KUKA KRL program: MyProgram_221().src

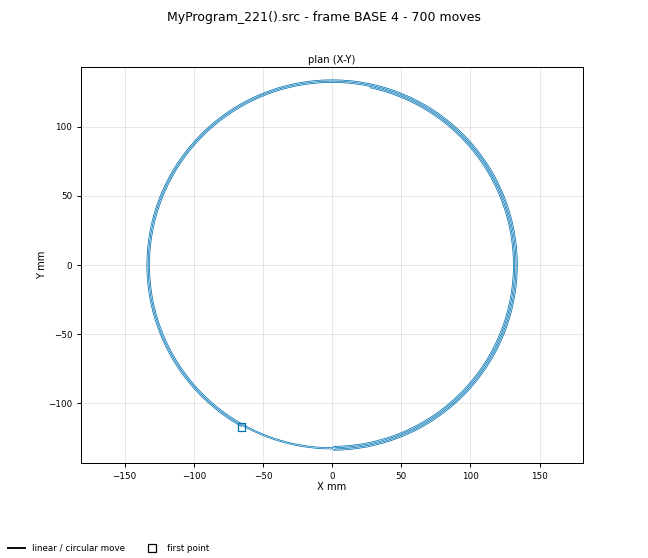
[picture p0: tool path of MyProgram_221().src in frame BASE 4, 700 of 700 moves have a stored position in this frame; points joined in program order, loops and branches not executed]
&ACCESS RVP
&REL 1
&PARAM TEMPLATE = C:\KRC\Roboter\Template\vorgabe
&PARAM EDITMASK = *
DEF MyProgram_221()
; ---- Setting reference (Base) ----
$BASE = BASE_DATA[4]

; --------------------------
; ---- Setting tool (TCP) ----
$TOOL = TOOL_DATA[3]
; --------------------------

$VEL.CP = VEL_APROX_PRINT
Startdeposition()
$VEL.CP = VEL_PRINT
LIN {X -65.4764,Y -116.7395,Z 154,A -122.5676,B 24.2106,C -1.1477,E1 24.1569,E2 209.4417} C_DIS
LIN {X -69.4702,Y -114.408,Z 154,A -124.5396,B 24.2105,C -1.151,E1 24.1522,E2 211.4118} C_DIS
LIN {X -73.2404,Y -112.0324,Z 154,A -126.4311,B 24.2103,C -1.1548,E1 24.1478,E2 213.3004} C_DIS
LIN {X -76.6718,Y -109.7121,Z 154,A -128.2386,B 24.2103,C -1.1561,E1 24.1436,E2 215.111} C_DIS
LIN {X -80.258,Y -107.117,Z 154,A -130.1581,B 24.2101,C -1.1583,E1 24.1393,E2 217.0323} C_DIS
LIN {X -83.7739,Y -104.39,Z 154,A -132.0662,B 24.21,C -1.1616,E1 24.1351,E2 218.9394} C_DIS
LIN {X -87.1638,Y -101.5764,Z 154,A -133.9639,B 24.2098,C -1.1647,E1 24.131,E2 220.837} C_DIS
LIN {X -90.549,Y -98.5704,Z 154,A -136.3247,B 24.2106,C -1.1484,E1 24.1261,E2 223.2477} C_DIS
LIN {X -93.7846,Y -95.4971,Z 154,A -138.0959,B 24.2101,C -1.1591,E1 24.1226,E2 225.0003} C_DIS
LIN {X -96.4017,Y -92.8551,Z 154,A -139.4034,B 24.2093,C -1.1762,E1 24.1201,E2 226.2717} C_DIS
LIN {X -99.4158,Y -89.621,Z 154,A -141.3271,B 24.2092,C -1.179,E1 24.1165,E2 228.1973} C_DIS
LIN {X -102.4018,Y -86.1925,Z 154,A -143.0746,B 24.2085,C -1.1931,E1 24.1133,E2 229.9185} C_DIS
LIN {X -107.1454,Y -80.2198,Z 154,A -146.5875,B 24.2087,C -1.1892,E1 24.1072,E2 233.4581} C_DIS
LIN {X -109.8326,Y -76.4986,Z 154,A -148.5307,B 24.2084,C -1.1953,E1 24.1041,E2 235.3964} C_DIS
LIN {X -112.3217,Y -72.7948,Z 154,A -150.4236,B 24.2082,C -1.2011,E1 24.1012,E2 237.2849} C_DIS
LIN {X -114.6316,Y -69.1005,Z 154,A -152.3129,B 24.208,C -1.2049,E1 24.0984,E2 239.1748} C_DIS
LIN {X -116.8933,Y -65.2026,Z 154,A -154.2587,B 24.2078,C -1.2094,E1 24.0957,E2 241.12} C_DIS
LIN {X -118.9758,Y -61.3183,Z 154,A -156.1666,B 24.2076,C -1.2137,E1 24.0933,E2 243.0279} C_DIS
LIN {X -120.9571,Y -57.3088,Z 154,A -158.0095,B 24.2072,C -1.2226,E1 24.091,E2 244.8594} C_DIS
LIN {X -122.9724,Y -52.8453,Z 154,A -160.0801,B 24.2068,C -1.2299,E1 24.0887,E2 246.9239} C_DIS
LIN {X -124.2089,Y -49.8691,Z 154,A -161.4613,B 24.2066,C -1.2339,E1 24.0872,E2 248.3033} C_DIS
LIN {X -125.3493,Y -46.9286,Z 154,A -162.8567,B 24.2066,C -1.2358,E1 24.0858,E2 249.702} C_DIS
LIN {X -126.5669,Y -43.5392,Z 154,A -164.3642,B 24.2062,C -1.2421,E1 24.0844,E2 251.2031} C_DIS
LIN {X -127.5513,Y -40.5643,Z 154,A -165.7297,B 24.2061,C -1.2451,E1 24.0833,E2 252.5694} C_DIS
LIN {X -128.4924,Y -37.4767,Z 154,A -167.1511,B 24.206,C -1.2475,E1 24.0821,E2 253.9935} C_DIS
LIN {X -129.5708,Y -33.5652,Z 154,A -169.0376,B 24.206,C -1.2458,E1 24.0807,E2 255.8954} C_DIS
LIN {X -130.5475,Y -29.5336,Z 154,A -170.6264,B 24.2054,C -1.2602,E1 24.0797,E2 257.4585} C_DIS
LIN {X -131.1874,Y -26.546,Z 154,A -172.5665,B 24.2066,C -1.2349,E1 24.0786,E2 259.4727} C_DIS
LIN {X -132.0312,Y -21.968,Z 154,A -173.9924,B 24.205,C -1.2676,E1 24.078,E2 260.827} C_DIS
LIN {X -132.553,Y -18.5652,Z 154,A -175.5736,B 24.205,C -1.2673,E1 24.0773,E2 262.4186} C_DIS
LIN {X -133.0698,Y -14.3967,Z 154,A -177.3185,B 24.2046,C -1.2756,E1 24.0768,E2 264.154} C_DIS
LIN {X -133.4458,Y -10.3664,Z 154,A -179.1414,B 24.2046,C -1.277,E1 24.0763,E2 265.9848} C_DIS
LIN {X -133.6901,Y -6.4724,Z 154,A 179.2809,B 24.204,C -1.2868,E1 24.0761,E2 267.5484} C_DIS
LIN {X -133.8245,Y -2.4362,Z 154,A 177.4846,B 24.204,C -1.2893,E1 24.076,E2 269.3498} C_DIS
LIN {X -133.831,Y 2.0454,Z 154,A 175.6023,B 24.2035,C -1.2973,E1 24.076,E2 271.2242} C_DIS
LIN {X -133.7281,Y 5.6424,Z 154,A 173.9321,B 24.2035,C -1.2963,E1 24.0762,E2 272.9073} C_DIS
LIN {X -133.4911,Y 9.7453,Z 154,A 172.2639,B 24.2031,C -1.3063,E1 24.0765,E2 274.5613} C_DIS
LIN {X -133.1347,Y 13.7941,Z 154,A 170.4691,B 24.2029,C -1.3094,E1 24.0769,E2 276.3596} C_DIS
LIN {X -132.7029,Y 17.4579,Z 154,A 168.9226,B 24.2026,C -1.3162,E1 24.0775,E2 277.8992} C_DIS
LIN {X -132.1182,Y 21.4462,Z 154,A 166.9905,B 24.2028,C -1.3122,E1 24.0783,E2 279.8529} C_DIS
LIN {X -131.3493,Y 25.7398,Z 154,A 165.3027,B 24.202,C -1.3266,E1 24.0792,E2 281.5157} C_DIS
LIN {X -129.9408,Y 32.1056,Z 154,A 162.5341,B 24.2015,C -1.3367,E1 24.0809,E2 284.2764} C_DIS
LIN {X -128.8361,Y 36.2779,Z 154,A 160.6208,B 24.2013,C -1.3396,E1 24.0823,E2 286.1942} C_DIS
LIN {X -127.7534,Y 39.9286,Z 154,A 158.5002,B 24.2023,C -1.322,E1 24.0841,E2 288.3705} C_DIS
LIN {X -126.4374,Y 43.913,Z 154,A 157.192,B 24.2008,C -1.3503,E1 24.0852,E2 289.6168} C_DIS
LIN {X -125.2818,Y 47.1088,Z 154,A 155.7275,B 24.2006,C -1.3544,E1 24.0866,E2 291.0799} C_DIS
LIN {X -124.0765,Y 50.1976,Z 154,A 154.2876,B 24.2004,C -1.3579,E1 24.0881,E2 292.5196} C_DIS
LIN {X -122.5281,Y 53.8719,Z 154,A 152.4761,B 24.2004,C -1.3583,E1 24.0901,E2 294.3407} C_DIS
LIN {X -119.6547,Y 59.9846,Z 154,A 149.6779,B 24.1997,C -1.3714,E1 24.0935,E2 297.1224} C_DIS
LIN {X -117.7054,Y 63.7246,Z 154,A 147.8801,B 24.1994,C -1.3771,E1 24.0958,E2 298.9159} C_DIS
LIN {X -116.2233,Y 66.3882,Z 154,A 146.4488,B 24.1994,C -1.3751,E1 24.0978,E2 300.3601} C_DIS
LIN {X -113.8859,Y 70.3235,Z 154,A 144.4779,B 24.1992,C -1.3802,E1 24.1006,E2 302.3289} C_DIS
LIN {X -111.5508,Y 73.9718,Z 154,A 142.5696,B 24.1991,C -1.383,E1 24.1035,E2 304.2403} C_DIS
LIN {X -108.9939,Y 77.6892,Z 154,A 140.6453,B 24.1987,C -1.3887,E1 24.1066,E2 306.1603} C_DIS
LIN {X -106.2792,Y 81.3632,Z 154,A 138.6861,B 24.1985,C -1.3939,E1 24.1099,E2 308.1166} C_DIS
LIN {X -103.8356,Y 84.4601,Z 154,A 136.9688,B 24.1983,C -1.3971,E1 24.1129,E2 309.8344} C_DIS
LIN {X -101.0139,Y 87.8152,Z 154,A 134.9381,B 24.1984,C -1.3947,E1 24.1166,E2 311.8804} C_DIS
LIN {X -96.0669,Y 93.2009,Z 154,A 131.9703,B 24.1976,C -1.4103,E1 24.1222,E2 314.8235} C_DIS
LIN {X -91.6081,Y 97.5874,Z 154,A 129.3779,B 24.197,C -1.4208,E1 24.1274,E2 317.4014} C_DIS
LIN {X -87.1976,Y 101.5473,Z 154,A 126.7888,B 24.1968,C -1.4242,E1 24.1328,E2 319.9928} C_DIS
LIN {X -84.1281,Y 104.1044,Z 154,A 124.7816,B 24.1974,C -1.4139,E1 24.1372,E2 322.033} C_DIS
LIN {X -81.4973,Y 106.1766,Z 154,A 123.2234,B 24.1975,C -1.4111,E1 24.1407,E2 323.604} C_DIS
LIN {X -78.3223,Y 108.54,Z 154,A 121.9651,B 24.1962,C -1.4353,E1 24.1434,E2 324.8076} C_DIS
LIN {X -75.2508,Y 110.6916,Z 154,A 120.2271,B 24.1964,C -1.4323,E1 24.1474,E2 326.5593} C_DIS
LIN {X -71.4037,Y 113.2111,Z 154,A 118.2937,B 24.1961,C -1.4377,E1 24.152,E2 328.4856} C_DIS
LIN {X -67.5784,Y 115.5356,Z 154,A 116.3255,B 24.196,C -1.4388,E1 24.1567,E2 330.4575} C_DIS
LIN {X -63.6092,Y 117.7676,Z 154,A 114.4022,B 24.1957,C -1.4434,E1 24.1614,E2 332.3751} C_DIS
LIN {X -60.562,Y 119.3608,Z 154,A 113.0252,B 24.1953,C -1.4505,E1 24.1648,E2 333.7388} C_DIS
LIN {X -57.5921,Y 120.8217,Z 154,A 111.5955,B 24.1953,C -1.4521,E1 24.1683,E2 335.1682} C_DIS
LIN {X -54.4903,Y 122.2521,Z 154,A 110.1144,B 24.1952,C -1.4535,E1 24.1721,E2 336.6499} C_DIS
LIN {X -51.3156,Y 123.6185,Z 154,A 108.6293,B 24.1951,C -1.4553,E1 24.1759,E2 338.1339} C_DIS
LIN {X -48.2296,Y 124.8548,Z 154,A 107.2262,B 24.1949,C -1.4583,E1 24.1796,E2 339.533} C_DIS
LIN {X -45.123,Y 126.0109,Z 154,A 105.7967,B 24.1949,C -1.4596,E1 24.1833,E2 340.9623} C_DIS
LIN {X -42.0962,Y 127.054,Z 154,A 104.423,B 24.1947,C -1.4611,E1 24.1869,E2 342.3349} C_DIS
LIN {X -38.7731,Y 128.1077,Z 154,A 102.9369,B 24.1947,C -1.4631,E1 24.1909,E2 343.8188} C_DIS
LIN {X -35.6125,Y 129.0222,Z 154,A 101.3601,B 24.195,C -1.4564,E1 24.1952,E2 345.4146} C_DIS
LIN {X -31.458,Y 130.0969,Z 154,A 99.6528,B 24.1945,C -1.4646,E1 24.1998,E2 347.1044} C_DIS
LIN {X -28.1162,Y 130.8598,Z 154,A 98.2044,B 24.1945,C -1.4668,E1 24.2037,E2 348.5493} C_DIS
LIN {X -24.9126,Y 131.5075,Z 154,A 96.7704,B 24.1945,C -1.4663,E1 24.2076,E2 349.9864} C_DIS
LIN {X -20.8025,Y 132.2202,Z 154,A 94.9726,B 24.1945,C -1.4669,E1 24.2126,E2 351.7842} C_DIS
LIN {X -17.2485,Y 132.7303,Z 154,A 93.4692,B 24.1943,C -1.4696,E1 24.2167,E2 353.2824} C_DIS
LIN {X -13.434,Y 133.172,Z 154,A 91.7062,B 24.1945,C -1.4646,E1 24.2217,E2 355.0588} C_DIS
LIN {X -9.6554,Y 133.4977,Z 154,A 90.2127,B 24.1941,C -1.4717,E1 24.2258,E2 356.5354} C_DIS
LIN {X -6.0046,Y 133.7136,Z 154,A 88.4886,B 24.1945,C -1.4644,E1 24.2306,E2 358.2778} C_DIS
LIN {X -2.0508,Y 133.8309,Z 154,A 86.9521,B 24.1941,C -1.4727,E1 24.2349,E2 359.7943} C_DIS
LIN {X 1.6346,Y 133.8378,Z 154,A 85.2383,B 24.1944,C -1.4661,E1 24.2397,E2 361.5239} C_DIS
LIN {X 5.3279,Y 133.7404,Z 154,A 83.7365,B 24.1942,C -1.4703,E1 24.2439,E2 363.0153} C_DIS
LIN {X 9.5685,Y 133.504,Z 154,A 81.9349,B 24.1942,C -1.4711,E1 24.2489,E2 364.8142} C_DIS
LIN {X 13.162,Y 133.1981,Z 154,A 80.3288,B 24.1944,C -1.4678,E1 24.2534,E2 366.4274} C_DIS
LIN {X 17.2746,Y 132.7269,Z 154,A 78.6281,B 24.1942,C -1.471,E1 24.2581,E2 368.1188} C_DIS
LIN {X 20.8308,Y 132.2158,Z 154,A 76.9846,B 24.1945,C -1.4652,E1 24.2626,E2 369.7748} C_DIS
LIN {X 24.9827,Y 131.4941,Z 154,A 75.2937,B 24.1942,C -1.4702,E1 24.2672,E2 371.4517} C_DIS
LIN {X 28.3093,Y 130.8181,Z 154,A 73.8631,B 24.1942,C -1.4706,E1 24.2711,E2 372.8794} C_DIS
LIN {X 31.4122,Y 130.1079,Z 154,A 72.501,B 24.1942,C -1.4699,E1 24.2748,E2 374.2414} C_DIS
LIN {X 34.6166,Y 129.2922,Z 154,A 71.066,B 24.1943,C -1.468,E1 24.2787,E2 375.6786} C_DIS
LIN {X 38.4085,Y 128.2193,Z 154,A 69.405,B 24.1943,C -1.468,E1 24.2832,E2 377.3366} C_DIS
LIN {X 40.9294,Y 127.4346,Z 154,A 67.9832,B 24.1952,C -1.4523,E1 24.2871,E2 378.7939} C_DIS
LIN {X 45.0326,Y 126.0435,Z 154,A 66.3563,B 24.1947,C -1.4622,E1 24.2913,E2 380.3933} C_DIS
LIN {X 48.6514,Y 124.6909,Z 154,A 64.7453,B 24.1947,C -1.4628,E1 24.2955,E2 381.9994} C_DIS
LIN {X 51.8882,Y 123.3793,Z 154,A 63.2634,B 24.1947,C -1.4618,E1 24.2993,E2 383.48} C_DIS
LIN {X 54.8155,Y 122.1066,Z 154,A 61.9074,B 24.1947,C -1.4608,E1 24.3027,E2 384.8351} C_DIS
LIN {X 57.9391,Y 120.656,Z 154,A 60.4143,B 24.1949,C -1.458,E1 24.3065,E2 386.331} C_DIS
LIN {X 61.0008,Y 119.1374,Z 154,A 58.9467,B 24.195,C -1.4558,E1 24.3102,E2 387.7997} C_DIS
LIN {X 64.4312,Y 117.3201,Z 154,A 57.1908,B 24.1954,C -1.4487,E1 24.3145,E2 389.5679} C_DIS
LIN {X 68.3558,Y 115.0772,Z 154,A 55.2802,B 24.1955,C -1.447,E1 24.3191,E2 391.4764} C_DIS
LIN {X 72.1374,Y 112.745,Z 154,A 53.3962,B 24.1956,C -1.445,E1 24.3236,E2 393.3591} C_DIS
LIN {X 76.0047,Y 110.1754,Z 154,A 51.4174,B 24.1958,C -1.4421,E1 24.3282,E2 395.3381} C_DIS
LIN {X 79.603,Y 107.6047,Z 154,A 49.5047,B 24.1961,C -1.4377,E1 24.3325,E2 397.2545} C_DIS
LIN {X 83.1317,Y 104.9021,Z 154,A 47.6134,B 24.1962,C -1.4347,E1 24.3367,E2 399.1457} C_DIS
LIN {X 86.5146,Y 102.1299,Z 154,A 45.7441,B 24.1964,C -1.4312,E1 24.3407,E2 401.016} C_DIS
LIN {X 90.0812,Y 98.9983,Z 154,A 43.7918,B 24.1964,C -1.4312,E1 24.3447,E2 402.9602} C_DIS
LIN {X 93.2562,Y 96.0134,Z 154,A 41.8886,B 24.1967,C -1.4253,E1 24.3486,E2 404.8697} C_DIS
LIN {X 96.3903,Y 92.8669,Z 154,A 40.0021,B 24.1969,C -1.4219,E1 24.3523,E2 406.7563} C_DIS
LIN {X 99.4022,Y 89.636,Z 154,A 38.0957,B 24.1972,C -1.4167,E1 24.3559,E2 408.6665} C_DIS
LIN {X 102.3288,Y 86.2796,Z 154,A 36.1869,B 24.1975,C -1.4121,E1 24.3593,E2 410.5776} C_DIS
LIN {X 105.1722,Y 82.7894,Z 154,A 34.2937,B 24.1976,C -1.4092,E1 24.3626,E2 412.4687} C_DIS
LIN {X 107.9981,Y 79.0677,Z 154,A 32.3149,B 24.1978,C -1.4053,E1 24.366,E2 414.4471} C_DIS
LIN {X 110.604,Y 75.3803,Z 154,A 30.3557,B 24.1982,C -1.3989,E1 24.3691,E2 416.4118} C_DIS
LIN {X 113.0003,Y 71.7377,Z 154,A 28.5033,B 24.1984,C -1.3947,E1 24.3719,E2 418.2649} C_DIS
LIN {X 115.3895,Y 67.8271,Z 154,A 26.5837,B 24.1986,C -1.3916,E1 24.3746,E2 420.1817} C_DIS
LIN {X 117.6737,Y 63.7829,Z 154,A 24.5746,B 24.1989,C -1.385,E1 24.3774,E2 422.1961} C_DIS
LIN {X 119.4521,Y 60.3826,Z 154,A 23.0754,B 24.1988,C -1.388,E1 24.3793,E2 423.6797} C_DIS
LIN {X 120.9911,Y 57.2375,Z 154,A 21.6009,B 24.1989,C -1.385,E1 24.3811,E2 425.1533} C_DIS
LIN {X 122.3009,Y 54.3811,Z 154,A 20.2749,B 24.1991,C -1.3821,E1 24.3826,E2 426.4788} C_DIS
LIN {X 123.551,Y 51.4772,Z 154,A 18.9001,B 24.1994,C -1.377,E1 24.3841,E2 427.8582} C_DIS
LIN {X 124.8078,Y 48.3505,Z 154,A 17.4767,B 24.1995,C -1.3737,E1 24.3855,E2 429.2814} C_DIS
LIN {X 125.9619,Y 45.259,Z 154,A 16.052,B 24.1998,C -1.3688,E1 24.3869,E2 430.7098} C_DIS
LIN {X 127.2555,Y 41.4902,Z 154,A 14.2466,B 24.2004,C -1.3582,E1 24.3885,E2 432.5303} C_DIS
LIN {X 128.9363,Y 35.9197,Z 154,A 11.8875,B 24.2004,C -1.3576,E1 24.3904,E2 434.8769} C_DIS
LIN {X 129.768,Y 32.7884,Z 154,A 10.5167,B 24.2006,C -1.3541,E1 24.3913,E2 436.248} C_DIS
LIN {X 130.6643,Y 29.0216,Z 154,A 8.745,B 24.2012,C -1.3427,E1 24.3925,E2 438.0367} C_DIS
LIN {X 131.466,Y 25.1297,Z 154,A 7.1682,B 24.2012,C -1.344,E1 24.3933,E2 439.6009} C_DIS
LIN {X 132.0838,Y 21.6522,Z 154,A 5.5745,B 24.2016,C -1.3347,E1 24.3941,E2 441.2073} C_DIS
LIN {X 132.7029,Y 17.4579,Z 154,A 3.892,B 24.2016,C -1.336,E1 24.3947,E2 442.8765} C_DIS
LIN {X 133.0904,Y 14.2054,Z 154,A 2.4559,B 24.2019,C -1.3296,E1 24.3952,E2 444.3193} C_DIS
LIN {X 133.4757,Y 9.9561,Z 154,A 0.6383,B 24.2021,C -1.3242,E1 24.3956,E2 446.1389} C_DIS
LIN {X 133.7017,Y 6.2399,Z 154,A -1.0342,B 24.2026,C -1.3147,E1 24.3958,E2 447.8241} C_DIS
LIN {X 133.8279,Y 2.2265,Z 154,A -2.6267,B 24.2026,C -1.3159,E1 24.3959,E2 449.4038} C_DIS
LIN {X 133.827,Y -2.2817,Z 154,A -4.5411,B 24.2028,C -1.3104,E1 24.3959,E2 451.3199} C_DIS
LIN {X 133.7017,Y -6.2409,Z 154,A -6.2871,B 24.2033,C -1.3021,E1 24.3957,E2 453.0752} C_DIS
LIN {X 133.4669,Y -10.0773,Z 154,A -7.9854,B 24.2037,C -1.2938,E1 24.3954,E2 454.7832} C_DIS
LIN {X 133.0839,Y -14.2661,Z 154,A -9.6488,B 24.2037,C -1.2953,E1 24.3949,E2 456.4328} C_DIS
LIN {X 132.6455,Y -17.8961,Z 154,A -11.2817,B 24.2041,C -1.2865,E1 24.3944,E2 458.0771} C_DIS
LIN {X 132.0424,Y -21.9007,Z 154,A -12.9201,B 24.2041,C -1.2859,E1 24.3936,E2 459.7068} C_DIS
LIN {X 131.4343,Y -25.2954,Z 154,A -14.392,B 24.2043,C -1.2813,E1 24.3929,E2 461.1809} C_DIS
LIN {X 130.5919,Y -29.3391,Z 154,A -16.2195,B 24.2048,C -1.2724,E1 24.3918,E2 463.0192} C_DIS
LIN {X 129.7273,Y -32.9487,Z 154,A -17.7013,B 24.2048,C -1.273,E1 24.3908,E2 464.4905} C_DIS
LIN {X 128.8805,Y -36.1191,Z 154,A -19.1001,B 24.2049,C -1.2688,E1 24.3898,E2 465.8912} C_DIS
LIN {X 127.9769,Y -39.2006,Z 154,A -20.4591,B 24.2051,C -1.2652,E1 24.3887,E2 467.2509} C_DIS
LIN {X 126.9685,Y -42.3527,Z 154,A -21.8818,B 24.2053,C -1.2604,E1 24.3875,E2 468.6769} C_DIS
LIN {X 125.8624,Y -45.5349,Z 154,A -23.3331,B 24.2056,C -1.2553,E1 24.3861,E2 470.1322} C_DIS
LIN {X 124.6655,Y -48.7165,Z 154,A -24.7733,B 24.2058,C -1.2515,E1 24.3847,E2 471.5731} C_DIS
LIN {X 123.3921,Y -51.8577,Z 154,A -26.187,B 24.2058,C -1.249,E1 24.3832,E2 472.9849} C_DIS
LIN {X 122.0866,Y -54.8603,Z 154,A -27.598,B 24.2061,C -1.2442,E1 24.3816,E2 474.3997} C_DIS
LIN {X 120.6489,Y -57.9539,Z 154,A -29.0501,B 24.2063,C -1.2401,E1 24.3798,E2 475.8535} C_DIS
LIN {X 118.8954,Y -61.476,Z 154,A -30.8726,B 24.2069,C -1.2275,E1 24.3775,E2 477.6965} C_DIS
LIN {X 116.6229,Y -65.6838,Z 154,A -32.8418,B 24.207,C -1.2256,E1 24.3749,E2 479.6597} C_DIS
LIN {X 114.3492,Y -69.5675,Z 154,A -34.7839,B 24.2073,C -1.2191,E1 24.3721,E2 481.6072} C_DIS
LIN {X 111.0229,Y -74.7614,Z 154,A -37.0916,B 24.2068,C -1.2294,E1 24.3686,E2 483.8781} C_DIS
LIN {X 105.8595,Y -81.9087,Z 154,A -41.023,B 24.2077,C -1.2103,E1 24.3622,E2 487.8361} C_DIS
LIN {X 104.1769,Y -84.0382,Z 154,A -42.2814,B 24.2081,C -1.202,E1 24.3599,E2 489.1085} C_DIS
LIN {X 101.5085,Y -87.2427,Z 154,A -44.0724,B 24.2084,C -1.197,E1 24.3567,E2 490.9033} C_DIS
LIN {X 98.4682,Y -90.6602,Z 154,A -46.0035,B 24.2085,C -1.1933,E1 24.3531,E2 492.8343} C_DIS
LIN {X 95.354,Y -93.9305,Z 154,A -47.9327,B 24.2088,C -1.1887,E1 24.3493,E2 494.7663} C_DIS
LIN {X 92.1619,Y -97.065,Z 154,A -49.8762,B 24.209,C -1.1825,E1 24.3454,E2 496.7165} C_DIS
LIN {X 88.9125,Y -100.0496,Z 154,A -51.7472,B 24.2092,C -1.1789,E1 24.3415,E2 498.5883} C_DIS
LIN {X 85.5504,Y -102.939,Z 154,A -53.5798,B 24.2092,C -1.178,E1 24.3376,E2 500.4157} C_DIS
LIN {X 82.3285,Y -105.534,Z 154,A -55.3614,B 24.2094,C -1.1735,E1 24.3337,E2 502.2013} C_DIS
LIN {X 78.8779,Y -108.1374,Z 154,A -57.2546,B 24.2097,C -1.1673,E1 24.3294,E2 504.1026} C_DIS
LIN {X 75.728,Y -110.3654,Z 154,A -58.6124,B 24.2092,C -1.1795,E1 24.3264,E2 505.426} C_DIS
LIN {X 73.182,Y -112.0704,Z 154,A -60.3562,B 24.2103,C -1.154,E1 24.3222,E2 507.2257} C_DIS
LIN {X 70.4805,Y -113.7885,Z 154,A -61.5128,B 24.2099,C -1.1626,E1 24.3195,E2 508.3576} C_DIS
LIN {X 65.7182,Y -116.6036,Z 154,A -63.893,B 24.2102,C -1.1576,E1 24.3138,E2 510.7425} C_DIS
LIN {X 61.9846,Y -118.6284,Z 154,A -65.5891,B 24.21,C -1.1609,E1 24.3096,E2 512.4256} C_DIS
LIN {X 59.0041,Y -120.1386,Z 154,A -67.0239,B 24.2101,C -1.1583,E1 24.306,E2 513.8628} C_DIS
LIN {X 55.9894,Y -121.5728,Z 154,A -68.4473,B 24.2102,C -1.1563,E1 24.3024,E2 515.2872} C_DIS
LIN {X 52.9146,Y -122.9424,Z 154,A -69.8817,B 24.2103,C -1.1544,E1 24.2988,E2 516.7225} C_DIS
LIN {X 49.7515,Y -124.2563,Z 154,A -71.3432,B 24.2103,C -1.1526,E1 24.295,E2 518.1852} C_DIS
LIN {X 46.4401,Y -125.5323,Z 154,A -72.8358,B 24.2104,C -1.1518,E1 24.2911,E2 519.6762} C_DIS
LIN {X 43.7144,Y -126.5062,Z 154,A -74.1092,B 24.2106,C -1.1484,E1 24.2877,E2 520.9552} C_DIS
LIN {X 40.4459,Y -127.5891,Z 154,A -75.5664,B 24.2106,C -1.1475,E1 24.2838,E2 522.4119} C_DIS
LIN {X 36.4957,Y -128.7752,Z 154,A -77.7145,B 24.2116,C -1.1257,E1 24.278,E2 524.6093} C_DIS
LIN {X 32.9651,Y -129.7231,Z 154,A -78.8975,B 24.2108,C -1.1438,E1 24.2749,E2 525.7463} C_DIS
LIN {X 29.7002,Y -130.5094,Z 154,A -80.3332,B 24.2108,C -1.1425,E1 24.271,E2 527.183} C_DIS
LIN {X 25.8378,Y -131.3306,Z 154,A -82.144,B 24.2112,C -1.1348,E1 24.266,E2 529.0104} C_DIS
LIN {X 22.0445,Y -132.0184,Z 154,A -83.6404,B 24.2109,C -1.1414,E1 24.2619,E2 530.4889} C_DIS
LIN {X 18.9624,Y -132.4962,Z 154,A -84.9944,B 24.2109,C -1.1395,E1 24.2582,E2 531.8463} C_DIS
LIN {X 15.267,Y -132.9741,Z 154,A -86.7055,B 24.2113,C -1.1325,E1 24.2534,E2 533.5731} C_DIS
LIN {X 11.3043,Y -133.3681,Z 154,A -88.2962,B 24.2111,C -1.1375,E1 24.249,E2 535.1507} C_DIS
LIN {X 7.55,Y -133.635,Z 154,A -90.0209,B 24.2114,C -1.1309,E1 24.2441,E2 536.8905} C_DIS
LIN {X 3.6306,Y -133.7972,Z 154,A -91.5862,B 24.2111,C -1.1362,E1 24.2398,E2 538.4427} C_DIS
LIN {X 0.9477,Y -133.839,Z 154,A -92.5277,B 24.2107,C -1.1466,E1 24.2373,E2 539.3588} C_DIS
Enddeposition()
LIN {X 0.9477,Y -133.839,Z 154,A -92.5277,B 24.2107,C -1.1466,E1 24.2373,E2 539.3588} C_DIS
Startdeposition()
$VEL.CP = VEL_PRINT
LIN {X 2.1127,Y -132.892,Z 154,A -91.1473,B 22.8975,C -0.9506,E1 22.9201,E2 538.3075} C_DIS
LIN {X 5.957,Y -132.7771,Z 154,A -89.4258,B 22.8973,C -0.9543,E1 22.925,E2 536.5772} C_DIS
LIN {X 9.4715,Y -132.5709,Z 154,A -88.025,B 22.8975,C -0.9493,E1 22.9288,E2 535.1899} C_DIS
LIN {X 12.5294,Y -132.3169,Z 154,A -86.6728,B 22.8975,C -0.9514,E1 22.9326,E2 533.8331} C_DIS
LIN {X 15.801,Y -131.966,Z 154,A -85.2691,B 22.8975,C -0.9514,E1 22.9365,E2 532.4303} C_DIS
LIN {X 19.2104,Y -131.5136,Z 154,A -83.7732,B 22.8974,C -0.9531,E1 22.9406,E2 530.9317} C_DIS
LIN {X 23.2039,Y -130.8675,Z 154,A -82.0552,B 22.8974,C -0.9531,E1 22.9454,E2 529.2155} C_DIS
LIN {X 27.7356,Y -129.9827,Z 154,A -80.0391,B 22.8973,C -0.9561,E1 22.9509,E2 527.1947} C_DIS
LIN {X 30.9445,Y -129.2561,Z 154,A -78.7716,B 22.8975,C -0.95,E1 22.9543,E2 525.9446} C_DIS
LIN {X 34.0346,Y -128.477,Z 154,A -77.2753,B 22.8972,C -0.9574,E1 22.9584,E2 524.4318} C_DIS
LIN {X 37.1351,Y -127.6153,Z 154,A -75.8896,B 22.8972,C -0.9589,E1 22.9621,E2 523.045} C_DIS
LIN {X 41.2179,Y -126.3581,Z 154,A -74.0508,B 22.8971,C -0.9609,E1 22.967,E2 521.2048} C_DIS
LIN {X 44.7886,Y -125.1347,Z 154,A -72.4048,B 22.897,C -0.9639,E1 22.9714,E2 519.5546} C_DIS
LIN {X 47.7741,Y -124.0259,Z 154,A -71.0402,B 22.897,C -0.9653,E1 22.9749,E2 518.1896} C_DIS
LIN {X 50.7753,Y -122.8279,Z 154,A -69.6151,B 22.8968,C -0.9689,E1 22.9786,E2 516.759} C_DIS
LIN {X 54.0596,Y -121.4175,Z 154,A -68.1256,B 22.8968,C -0.9687,E1 22.9824,E2 515.2741} C_DIS
LIN {X 57.0881,Y -120.0233,Z 154,A -66.7624,B 22.8968,C -0.9672,E1 22.9859,E2 513.9183} C_DIS
LIN {X 59.7376,Y -118.7283,Z 154,A -65.508,B 22.8968,C -0.9684,E1 22.989,E2 512.6646} C_DIS
LIN {X 63.0059,Y -117.0273,Z 154,A -63.7534,B 22.8963,C -0.9795,E1 22.9934,E2 510.8873} C_DIS
LIN {X 66.9552,Y -114.8142,Z 154,A -61.8237,B 22.8963,C -0.9818,E1 22.9981,E2 508.9578} C_DIS
LIN {X 70.582,Y -112.6209,Z 154,A -59.9604,B 22.896,C -0.9871,E1 23.0025,E2 507.0875} C_DIS
LIN {X 74.255,Y -110.2334,Z 154,A -58.154,B 22.896,C -0.9867,E1 23.0067,E2 505.2888} C_DIS
LIN {X 77.655,Y -107.8656,Z 154,A -56.3006,B 22.8958,C -0.9937,E1 23.0109,E2 503.4245} C_DIS
LIN {X 81.0836,Y -105.3126,Z 154,A -54.453,B 22.8956,C -0.9979,E1 23.0151,E2 501.5736} C_DIS
LIN {X 84.5996,Y -102.5089,Z 154,A -52.5864,B 22.8956,C -0.9985,E1 23.0191,E2 499.7132} C_DIS
LIN {X 87.7093,Y -99.8618,Z 154,A -50.7833,B 22.8953,C -1.0047,E1 23.0229,E2 497.9021} C_DIS
LIN {X 90.8925,Y -96.9735,Z 154,A -48.9399,B 22.8951,C -1.0086,E1 23.0267,E2 496.057} C_DIS
LIN {X 94.0651,Y -93.8987,Z 154,A -47.0483,B 22.895,C -1.0126,E1 23.0305,E2 494.1641} C_DIS
LIN {X 97.1866,Y -90.6636,Z 154,A -45.1477,B 22.8949,C -1.0155,E1 23.0341,E2 492.265} C_DIS
LIN {X 100.0672,Y -87.4738,Z 154,A -43.306,B 22.8947,C -1.0197,E1 23.0375,E2 490.4218} C_DIS
LIN {X 102.9883,Y -84.0151,Z 154,A -41.4128,B 22.8946,C -1.0218,E1 23.0409,E2 488.5327} C_DIS
LIN {X 105.6436,Y -80.6507,Z 154,A -39.5771,B 22.8944,C -1.0262,E1 23.044,E2 486.6954} C_DIS
LIN {X 108.0483,Y -77.3995,Z 154,A -37.7996,B 22.8941,C -1.0327,E1 23.047,E2 484.9106} C_DIS
LIN {X 110.6056,Y -73.6989,Z 154,A -35.9199,B 22.8941,C -1.0351,E1 23.0499,E2 483.035} C_DIS
LIN {X 112.7841,Y -70.3198,Z 154,A -34.1534,B 22.8937,C -1.0418,E1 23.0526,E2 481.2614} C_DIS
LIN {X 115.1096,Y -66.4448,Z 154,A -32.2669,B 22.8937,C -1.0442,E1 23.0552,E2 479.3792} C_DIS
LIN {X 117.0273,Y -63.0059,Z 154,A -30.5354,B 22.8933,C -1.051,E1 23.0576,E2 477.6405} C_DIS
LIN {X 118.9136,Y -59.368,Z 154,A -28.8093,B 22.8932,C -1.0542,E1 23.0597,E2 475.9163} C_DIS
LIN {X 120.5049,Y -56.0647,Z 154,A -27.3043,B 22.8932,C -1.0551,E1 23.0615,E2 474.418} C_DIS
LIN {X 121.9041,Y -52.9532,Z 154,A -25.8432,B 22.893,C -1.0591,E1 23.0632,E2 472.9554} C_DIS
LIN {X 123.1105,Y -50.086,Z 154,A -24.6641,B 22.8932,C -1.0549,E1 23.0644,E2 471.7942} C_DIS
LIN {X 124.1759,Y -47.3882,Z 154,A -23.2722,B 22.8927,C -1.066,E1 23.0659,E2 470.3825} C_DIS
LIN {X 125.3771,Y -44.1087,Z 154,A -21.7006,B 22.8923,C -1.0741,E1 23.0673,E2 468.7998} C_DIS
LIN {X 126.3581,Y -41.2179,Z 154,A -20.4741,B 22.8923,C -1.0736,E1 23.0684,E2 467.5823} C_DIS
LIN {X 127.3266,Y -38.1213,Z 154,A -18.9442,B 22.8918,C -1.0848,E1 23.0697,E2 466.0334} C_DIS
LIN {X 128.3554,Y -34.4904,Z 154,A -17.4668,B 22.892,C -1.0823,E1 23.0708,E2 464.5717} C_DIS
LIN {X 129.1734,Y -31.2877,Z 154,A -16.1518,B 22.892,C -1.0812,E1 23.0716,E2 463.2678} C_DIS
LIN {X 129.8696,Y -28.2593,Z 154,A -14.7347,B 22.8916,C -1.0895,E1 23.0725,E2 461.8387} C_DIS
LIN {X 130.5311,Y -25.0263,Z 154,A -13.5237,B 22.8919,C -1.0832,E1 23.0732,E2 460.6515} C_DIS
LIN {X 131.0612,Y -22.0836,Z 154,A -12.0224,B 22.8912,C -1.0983,E1 23.0739,E2 459.1215} C_DIS
LIN {X 131.5475,Y -18.9729,Z 154,A -10.7202,B 22.8912,C -1.0998,E1 23.0744,E2 457.8238} C_DIS
LIN {X 131.9593,Y -15.8571,Z 154,A -9.3232,B 22.8909,C -1.1064,E1 23.0749,E2 456.4191} C_DIS
LIN {X 132.3732,Y -11.9426,Z 154,A -7.6777,B 22.8907,C -1.1092,E1 23.0754,E2 454.7771} C_DIS
LIN {X 132.6446,Y -8.3772,Z 154,A -6.129,B 22.8905,C -1.1146,E1 23.0757,E2 453.2247} C_DIS
LIN {X 132.8117,Y -5.08,Z 154,A -4.7083,B 22.8903,C -1.1191,E1 23.0759,E2 451.8018} C_DIS
LIN {X 132.9061,Y -0.9754,Z 154,A -3.2387,B 22.8907,C -1.1094,E1 23.0759,E2 450.3666} C_DIS
LIN {X 132.8937,Y 2.0094,Z 154,A -1.7075,B 22.89,C -1.1261,E1 23.0759,E2 448.8028} C_DIS
LIN {X 132.7482,Y 6.5315,Z 154,A 0.2582,B 22.8896,C -1.1332,E1 23.0757,E2 446.8319} C_DIS
LIN {X 132.5374,Y 9.9303,Z 154,A 1.7552,B 22.8893,C -1.1394,E1 23.0754,E2 445.3288} C_DIS
LIN {X 132.1681,Y 14.0127,Z 154,A 3.2376,B 22.8897,C -1.1305,E1 23.075,E2 443.8789} C_DIS
LIN {X 131.809,Y 17.0623,Z 154,A 4.8026,B 22.889,C -1.1471,E1 23.0745,E2 442.2818} C_DIS
LIN {X 131.3388,Y 20.3671,Z 154,A 6.2278,B 22.8888,C -1.1509,E1 23.0739,E2 440.856} C_DIS
LIN {X 130.6919,Y 24.1849,Z 154,A 7.8576,B 22.8886,C -1.1542,E1 23.0731,E2 439.2284} C_DIS
LIN {X 130.0822,Y 27.2746,Z 154,A 9.2079,B 22.8884,C -1.158,E1 23.0723,E2 437.8769} C_DIS
LIN {X 129.3944,Y 30.3708,Z 154,A 10.5676,B 22.8883,C -1.1619,E1 23.0715,E2 436.516} C_DIS
LIN {X 128.484,Y 34.0083,Z 154,A 12.1821,B 22.888,C -1.1668,E1 23.0704,E2 434.8991} C_DIS
LIN {X 127.6153,Y 37.1351,Z 154,A 13.5667,B 22.8879,C -1.1704,E1 23.0693,E2 433.5143} C_DIS
LIN {X 126.6727,Y 40.233,Z 154,A 14.7649,B 22.8881,C -1.1646,E1 23.0683,E2 432.3385} C_DIS
LIN {X 125.6807,Y 43.2328,Z 154,A 16.3339,B 22.8874,C -1.1792,E1 23.0669,E2 430.7419} C_DIS
LIN {X 124.5426,Y 46.409,Z 154,A 17.7686,B 22.8873,C -1.1825,E1 23.0656,E2 429.3075} C_DIS
LIN {X 123.3544,Y 49.4809,Z 154,A 19.0824,B 22.8873,C -1.1813,E1 23.0642,E2 428.0048} C_DIS
LIN {X 122.16,Y 52.3614,Z 154,A 20.4686,B 22.887,C -1.1873,E1 23.0627,E2 426.6115} C_DIS
LIN {X 120.9852,Y 55.0261,Z 154,A 21.7528,B 22.8868,C -1.1924,E1 23.0612,E2 425.3221} C_DIS
LIN {X 119.5649,Y 58.0477,Z 154,A 23.2927,B 22.8863,C -1.2016,E1 23.0594,E2 423.7679} C_DIS
LIN {X 118.0626,Y 61.0452,Z 154,A 24.7572,B 22.8861,C -1.2066,E1 23.0575,E2 422.2992} C_DIS
LIN {X 115.9198,Y 65.021,Z 154,A 26.6466,B 22.886,C -1.209,E1 23.0549,E2 420.4144} C_DIS
LIN {X 113.6134,Y 68.9721,Z 154,A 28.605,B 22.8857,C -1.2136,E1 23.0522,E2 418.4553} C_DIS
LIN {X 111.2458,Y 72.7301,Z 154,A 30.5578,B 22.8854,C -1.2206,E1 23.0492,E2 416.4956} C_DIS
LIN {X 108.8049,Y 76.333,Z 154,A 32.3426,B 22.8854,C -1.2208,E1 23.0464,E2 414.72} C_DIS
LIN {X 106.3485,Y 79.72,Z 154,A 34.2123,B 22.885,C -1.2286,E1 23.0433,E2 412.8402} C_DIS
LIN {X 103.7242,Y 83.1058,Z 154,A 35.9974,B 22.8849,C -1.23,E1 23.0402,E2 411.0607} C_DIS
LIN {X 100.9873,Y 86.411,Z 154,A 37.8811,B 22.8846,C -1.236,E1 23.0368,E2 409.171} C_DIS
LIN {X 98.1414,Y 89.6301,Z 154,A 39.7242,B 22.8844,C -1.2398,E1 23.0333,E2 407.3273} C_DIS
LIN {X 95.1345,Y 92.8152,Z 154,A 41.5798,B 22.8843,C -1.2423,E1 23.0297,E2 405.4741} C_DIS
LIN {X 92.1398,Y 95.7891,Z 154,A 43.3706,B 22.8841,C -1.2448,E1 23.0262,E2 403.6853} C_DIS
LIN {X 88.9934,Y 98.7191,Z 154,A 45.2552,B 22.8839,C -1.2501,E1 23.0223,E2 401.7954} C_DIS
LIN {X 85.6465,Y 101.636,Z 154,A 47.1272,B 22.8838,C -1.2518,E1 23.0183,E2 399.9271} C_DIS
LIN {X 82.4349,Y 104.2582,Z 154,A 48.942,B 22.8835,C -1.2565,E1 23.0144,E2 398.1078} C_DIS
LIN {X 78.9493,Y 106.9216,Z 154,A 50.823,B 22.8834,C -1.2595,E1 23.0102,E2 396.2268} C_DIS
LIN {X 75.3782,Y 109.4682,Z 154,A 52.6982,B 22.8832,C -1.2619,E1 23.0059,E2 394.3524} C_DIS
LIN {X 71.5466,Y 112.0099,Z 154,A 54.6437,B 22.8832,C -1.2633,E1 23.0013,E2 392.4104} C_DIS
LIN {X 67.7007,Y 114.3761,Z 154,A 56.5773,B 22.8831,C -1.2656,E1 22.9967,E2 390.4775} C_DIS
LIN {X 64.0155,Y 116.4788,Z 154,A 58.4069,B 22.8829,C -1.2682,E1 22.9922,E2 388.6472} C_DIS
LIN {X 61.0452,Y 118.0626,Z 154,A 59.9017,B 22.8827,C -1.2723,E1 22.9885,E2 387.1465} C_DIS
LIN {X 57.9811,Y 119.5967,Z 154,A 61.2114,B 22.883,C -1.266,E1 22.9853,E2 385.8568} C_DIS
LIN {X 54.7444,Y 121.1112,Z 154,A 62.7467,B 22.883,C -1.2676,E1 22.9814,E2 384.3217} C_DIS
LIN {X 51.4984,Y 122.526,Z 154,A 64.2739,B 22.8829,C -1.2694,E1 22.9775,E2 382.7941} C_DIS
LIN {X 48.3654,Y 123.796,Z 154,A 65.518,B 22.8833,C -1.2606,E1 22.9743,E2 381.5756} C_DIS
LIN {X 45.3862,Y 124.9193,Z 154,A 67.1241,B 22.8827,C -1.2732,E1 22.97,E2 379.941} C_DIS
LIN {X 42.2017,Y 126.0305,Z 154,A 68.3378,B 22.8832,C -1.2628,E1 22.9669,E2 378.7564} C_DIS
LIN {X 39.2935,Y 126.9678,Z 154,A 69.7269,B 22.883,C -1.2674,E1 22.9632,E2 377.3586} C_DIS
LIN {X 36.5715,Y 127.7803,Z 154,A 71.2479,B 22.8822,C -1.2825,E1 22.959,E2 375.8015} C_DIS
LIN {X 32.8287,Y 128.7903,Z 154,A 72.7455,B 22.8825,C -1.2753,E1 22.955,E2 374.3251} C_DIS
LIN {X 28.8221,Y 129.7481,Z 154,A 74.536,B 22.8825,C -1.2769,E1 22.9502,E2 372.533} C_DIS
LIN {X 25.4913,Y 130.4422,Z 154,A 76.0774,B 22.8822,C -1.2812,E1 22.9459,E2 370.9827} C_DIS
LIN {X 22.0622,Y 131.0648,Z 154,A 77.462,B 22.8825,C -1.2762,E1 22.9421,E2 369.6127} C_DIS
LIN {X 18.0354,Y 131.6815,Z 154,A 79.4068,B 22.882,C -1.2857,E1 22.9367,E2 367.6455} C_DIS
LIN {X 14.9807,Y 132.0639,Z 154,A 80.7296,B 22.882,C -1.2857,E1 22.9331,E2 366.3236} C_DIS
LIN {X 11.4569,Y 132.4142,Z 154,A 82.1227,B 22.8823,C -1.2796,E1 22.9292,E2 364.9472} C_DIS
LIN {X 8.2404,Y 132.653,Z 154,A 83.5325,B 22.8823,C -1.2806,E1 22.9253,E2 363.5355} C_DIS
LIN {X 4.4346,Y 132.8368,Z 154,A 85.1243,B 22.8824,C -1.278,E1 22.9209,E2 361.9508} C_DIS
LIN {X 0.8253,Y 132.9063,Z 154,A 86.7307,B 22.8823,C -1.2802,E1 22.9164,E2 360.3389} C_DIS
LIN {X -2.9501,Y 132.8781,Z 154,A 88.46,B 22.8821,C -1.2846,E1 22.9115,E2 358.5982} C_DIS
LIN {X -6.6414,Y 132.7427,Z 154,A 89.9475,B 22.8823,C -1.2792,E1 22.9074,E2 357.1242} C_DIS
LIN {X -10.4305,Y 132.5009,Z 154,A 91.5475,B 22.8825,C -1.2768,E1 22.9029,E2 355.5297} C_DIS
LIN {X -14.0127,Y 132.1681,Z 154,A 93.1282,B 22.8825,C -1.2775,E1 22.8985,E2 353.9464} C_DIS
LIN {X -17.0623,Y 131.809,Z 154,A 94.4706,B 22.8825,C -1.2775,E1 22.8948,E2 352.6027} C_DIS
LIN {X -20.2784,Y 131.3525,Z 154,A 95.7329,B 22.8828,C -1.2703,E1 22.8914,E2 351.3581} C_DIS
LIN {X -23.2039,Y 130.8675,Z 154,A 97.119,B 22.8826,C -1.2743,E1 22.8875,E2 349.96} C_DIS
LIN {X -27.2746,Y 130.0822,Z 154,A 98.9119,B 22.8826,C -1.2731,E1 22.8826,E2 348.1679} C_DIS
LIN {X -30.3708,Y 129.3944,Z 154,A 100.2841,B 22.8827,C -1.2721,E1 22.8789,E2 346.7964} C_DIS
LIN {X -33.9605,Y 128.4968,Z 154,A 101.922,B 22.8827,C -1.2726,E1 22.8745,E2 345.1547} C_DIS
LIN {X -37.1351,Y 127.6153,Z 154,A 103.3113,B 22.8828,C -1.2697,E1 22.8707,E2 343.7704} C_DIS
LIN {X -41.2179,Y 126.3581,Z 154,A 105.2985,B 22.8826,C -1.2743,E1 22.8654,E2 341.7676} C_DIS
LIN {X -44.8685,Y 125.1059,Z 154,A 106.8308,B 22.883,C -1.2662,E1 22.8614,E2 340.2528} C_DIS
LIN {X -47.3882,Y 124.1759,Z 154,A 107.9934,B 22.883,C -1.2648,E1 22.8584,E2 339.0909} C_DIS
LIN {X -50.4557,Y 122.9614,Z 154,A 109.4216,B 22.8832,C -1.2632,E1 22.8547,E2 337.6636} C_DIS
LIN {X -53.7849,Y 121.5404,Z 154,A 111.0381,B 22.8832,C -1.2635,E1 22.8505,E2 336.0421} C_DIS
LIN {X -57.0213,Y 120.0552,Z 154,A 112.4393,B 22.8836,C -1.255,E1 22.847,E2 334.6588} C_DIS
LIN {X -59.5497,Y 118.8239,Z 154,A 113.7488,B 22.8835,C -1.2575,E1 22.8437,E2 333.3391} C_DIS
LIN {X -63.0059,Y 117.0273,Z 154,A 115.5233,B 22.8834,C -1.2591,E1 22.8393,E2 331.5552} C_DIS
LIN {X -66.9552,Y 114.8142,Z 154,A 117.5244,B 22.8834,C -1.2579,E1 22.8345,E2 329.5506} C_DIS
LIN {X -70.7172,Y 112.5356,Z 154,A 119.4231,B 22.8836,C -1.2545,E1 22.83,E2 327.6541} C_DIS
LIN {X -74.5989,Y 110.0006,Z 154,A 121.3824,B 22.8839,C -1.2488,E1 22.8254,E2 325.7023} C_DIS
LIN {X -78.2784,Y 107.4138,Z 154,A 123.2692,B 22.8843,C -1.2425,E1 22.8212,E2 323.8245} C_DIS
LIN {X -81.5146,Y 104.9786,Z 154,A 125.0594,B 22.8843,C -1.2409,E1 22.8172,E2 322.0314} C_DIS
LIN {X -84.8863,Y 102.2714,Z 154,A 126.95,B 22.8845,C -1.238,E1 22.8131,E2 320.1404} C_DIS
LIN {X -88.119,Y 99.4996,Z 154,A 128.7793,B 22.8847,C -1.2336,E1 22.8092,E2 318.3146} C_DIS
LIN {X -91.2905,Y 96.5979,Z 154,A 130.6426,B 22.8849,C -1.2297,E1 22.8054,E2 316.4529} C_DIS
LIN {X -94.2026,Y 93.7602,Z 154,A 132.4531,B 22.8849,C -1.2281,E1 22.8018,E2 314.6382} C_DIS
LIN {X -97.1866,Y 90.6636,Z 154,A 134.3165,B 22.8852,C -1.2239,E1 22.7983,E2 312.7766} C_DIS
LIN {X -100.0672,Y 87.4738,Z 154,A 136.1797,B 22.8854,C -1.2197,E1 22.7948,E2 310.9151} C_DIS
LIN {X -103.0364,Y 83.9562,Z 154,A 138.1692,B 22.8857,C -1.2148,E1 22.7913,E2 308.9282} C_DIS
LIN {X -105.6436,Y 80.6507,Z 154,A 139.954,B 22.886,C -1.2086,E1 22.7882,E2 307.1501} C_DIS
LIN {X -108.1522,Y 77.2542,Z 154,A 141.7957,B 22.8862,C -1.2046,E1 22.7852,E2 305.3088} C_DIS
LIN {X -110.6644,Y 73.6107,Z 154,A 143.686,B 22.8865,C -1.1985,E1 22.7822,E2 303.4239} C_DIS
LIN {X -112.8996,Y 70.1342,Z 154,A 145.5296,B 22.8865,C -1.1962,E1 22.7795,E2 301.5758} C_DIS
LIN {X -115.0838,Y 66.4895,Z 154,A 147.3383,B 22.8869,C -1.1899,E1 22.7769,E2 299.7732} C_DIS
LIN {X -117.0273,Y 63.0059,Z 154,A 149.1139,B 22.887,C -1.1874,E1 22.7745,E2 297.9937} C_DIS
LIN {X -118.8239,Y 59.5497,Z 154,A 150.714,B 22.8874,C -1.1789,E1 22.7725,E2 296.4062} C_DIS
LIN {X -120.3608,Y 56.3764,Z 154,A 152.3326,B 22.8874,C -1.1787,E1 22.7706,E2 294.7784} C_DIS
LIN {X -121.9041,Y 52.9532,Z 154,A 153.871,B 22.8879,C -1.1703,E1 22.7689,E2 293.2524} C_DIS
LIN {X -122.9614,Y 50.4557,Z 154,A 155.1798,B 22.8877,C -1.1728,E1 22.7674,E2 291.929} C_DIS
LIN {X -124.3532,Y 46.9147,Z 154,A 156.7126,B 22.8882,C -1.163,E1 22.7659,E2 290.4119} C_DIS
LIN {X -125.5099,Y 43.7257,Z 154,A 158.1629,B 22.8884,C -1.158,E1 22.7646,E2 288.9657} C_DIS
LIN {X -126.8525,Y 39.6702,Z 154,A 160.0212,B 22.8887,C -1.1529,E1 22.763,E2 287.1088} C_DIS
LIN {X -127.7803,Y 36.5715,Z 154,A 161.424,B 22.8889,C -1.1489,E1 22.7619,E2 285.7074} C_DIS
LIN {X -128.7348,Y 33.0475,Z 154,A 163.0439,B 22.889,C -1.1459,E1 22.7607,E2 284.0847} C_DIS
LIN {X -129.3944,Y 30.3708,Z 154,A 164.2026,B 22.8893,C -1.1408,E1 22.76,E2 282.9318} C_DIS
LIN {X -130.0822,Y 27.2746,Z 154,A 165.5794,B 22.8895,C -1.1368,E1 22.7592,E2 281.5563} C_DIS
LIN {X -130.6919,Y 24.1849,Z 154,A 167.1042,B 22.8893,C -1.1399,E1 22.7584,E2 280.0138} C_DIS
LIN {X -131.2246,Y 21.1043,Z 154,A 168.461,B 22.8895,C -1.1359,E1 22.7578,E2 278.6583} C_DIS
LIN {X -131.6815,Y 18.0354,Z 154,A 169.8025,B 22.8897,C -1.1318,E1 22.7572,E2 277.3186} C_DIS
LIN {X -132.0639,Y 14.9807,Z 154,A 171.1358,B 22.8899,C -1.1277,E1 22.7568,E2 275.9869} C_DIS
LIN {X -132.3732,Y 11.9426,Z 154,A 172.4549,B 22.8901,C -1.1236,E1 22.7565,E2 274.6699} C_DIS
LIN {X -132.651,Y 8.2731,Z 154,A 173.9205,B 22.8906,C -1.1131,E1 22.7562,E2 273.2215} C_DIS
LIN {X -132.8178,Y 4.9227,Z 154,A 175.398,B 22.8907,C -1.1098,E1 22.756,E2 271.7428} C_DIS
LIN {X -132.9027,Y 1.4718,Z 154,A 176.7927,B 22.8911,C -1.1009,E1 22.756,E2 270.362} C_DIS
LIN {X -132.8937,Y -2.0094,Z 154,A 178.362,B 22.8911,C -1.0991,E1 22.756,E2 268.7869} C_DIS
LIN {X -132.7507,Y -6.4816,Z 154,A -179.6441,B 22.8913,C -1.0957,E1 22.7562,E2 266.7884} C_DIS
LIN {X -132.5709,Y -9.4715,Z 154,A -178.3869,B 22.8916,C -1.0901,E1 22.7564,E2 265.5376} C_DIS
LIN {X -132.1681,Y -14.0127,Z 154,A -176.6198,B 22.8923,C -1.075,E1 22.7569,E2 263.7976} C_DIS
LIN {X -131.809,Y -17.0623,Z 154,A -175.0675,B 22.892,C -1.0809,E1 22.7574,E2 262.22} C_DIS
LIN {X -131.2246,Y -21.1043,Z 154,A -173.1297,B 22.892,C -1.0831,E1 22.7582,E2 260.2635} C_DIS
LIN {X -130.3968,Y -25.7288,Z 154,A -171.2481,B 22.8925,C -1.0704,E1 22.7592,E2 258.4026} C_DIS
LIN {X -129.7481,Y -28.8221,Z 154,A -169.8738,B 22.8926,C -1.0667,E1 22.76,E2 257.029} C_DIS
LIN {X -128.9474,Y -32.2099,Z 154,A -168.2837,B 22.8926,C -1.066,E1 22.7611,E2 255.4303} C_DIS
LIN {X -128.0562,Y -35.585,Z 154,A -166.8419,B 22.893,C -1.0586,E1 22.7621,E2 253.9985} C_DIS
LIN {X -127.1542,Y -38.6846,Z 154,A -165.4384,B 22.8932,C -1.0549,E1 22.7632,E2 252.5956} C_DIS
LIN {X -126.2079,Y -41.6691,Z 154,A -164.0476,B 22.8932,C -1.0527,E1 22.7644,E2 251.2018} C_DIS
LIN {X -125.1059,Y -44.8685,Z 154,A -162.607,B 22.8935,C -1.0475,E1 22.7658,E2 249.7655} C_DIS
LIN {X -124.1759,Y -47.3882,Z 154,A -161.3222,B 22.8934,C -1.0497,E1 22.767,E2 248.467} C_DIS
LIN {X -122.7412,Y -50.983,Z 154,A -159.908,B 22.8941,C -1.0335,E1 22.7685,E2 247.086} C_DIS
LIN {X -121.4467,Y -53.9943,Z 154,A -158.316,B 22.8939,C -1.0374,E1 22.7703,E2 245.4743} C_DIS
LIN {X -120.0233,Y -57.0881,Z 154,A -156.8495,B 22.8941,C -1.0332,E1 22.772,E2 244.0099} C_DIS
LIN {X -118.5347,Y -60.1178,Z 154,A -155.4046,B 22.8943,C -1.0286,E1 22.7738,E2 242.5682} C_DIS
LIN {X -116.8823,Y -63.2757,Z 154,A -153.7664,B 22.8943,C -1.0289,E1 22.776,E2 240.9196} C_DIS
LIN {X -114.8052,Y -66.9704,Z 154,A -151.8827,B 22.8943,C -1.0265,E1 22.7786,E2 239.0313} C_DIS
LIN {X -112.5786,Y -70.649,Z 154,A -150.0367,B 22.8946,C -1.0213,E1 22.7813,E2 237.1884} C_DIS
LIN {X -110.3046,Y -74.1497,Z 154,A -148.1958,B 22.8947,C -1.0185,E1 22.7842,E2 235.3445} C_DIS
LIN {X -107.7937,Y -77.7542,Z 154,A -146.2963,B 22.8949,C -1.014,E1 22.7872,E2 233.4464} C_DIS
LIN {X -105.3126,Y -81.0836,Z 154,A -144.5409,B 22.8952,C -1.008,E1 22.7902,E2 231.6972} C_DIS
LIN {X -102.6401,Y -84.4411,Z 154,A -142.6255,B 22.8952,C -1.0066,E1 22.7936,E2 229.7757} C_DIS
LIN {X -99.8618,Y -87.7093,Z 154,A -140.7771,B 22.8954,C -1.0023,E1 22.7969,E2 227.9291} C_DIS
LIN {X -96.9735,Y -90.8925,Z 154,A -138.9142,B 22.8956,C -0.9986,E1 22.8005,E2 226.0667} C_DIS
LIN {X -93.9822,Y -93.9822,Z 154,A -137.0947,B 22.8958,C -0.993,E1 22.804,E2 224.253} C_DIS
LIN {X -90.8925,Y -96.9735,Z 154,A -135.232,B 22.8959,C -0.9896,E1 22.8078,E2 222.3907} C_DIS
LIN {X -87.7093,Y -99.8618,Z 154,A -133.3709,B 22.8961,C -0.9862,E1 22.8117,E2 220.5301} C_DIS
LIN {X -84.4379,Y -102.6428,Z 154,A -131.4688,B 22.8961,C -0.985,E1 22.8157,E2 218.6231} C_DIS
LIN {X -81.0836,Y -105.3126,Z 154,A -129.6571,B 22.8963,C -0.98,E1 22.8197,E2 216.817} C_DIS
LIN {X -77.6523,Y -107.8676,Z 154,A -127.7633,B 22.8963,C -0.9791,E1 22.824,E2 214.9183} C_DIS
LIN {X -74.0817,Y -110.35,Z 154,A -125.8816,B 22.8965,C -0.9763,E1 22.8283,E2 213.0367} C_DIS
LIN {X -70.3198,Y -112.7841,Z 154,A -123.9746,B 22.8966,C -0.9722,E1 22.8328,E2 211.1337} C_DIS
LIN {X -66.4895,Y -115.0838,Z 154,A -122.0845,B 22.8968,C -0.9677,E1 22.8374,E2 209.2489} C_DIS
LIN {X -63.0059,Y -117.0273,Z 154,A -120.2737,B 22.8968,C -0.9696,E1 22.8418,E2 207.4275} C_DIS
LIN {X -59.5497,Y -118.8239,Z 154,A -118.6143,B 22.8968,C -0.9665,E1 22.8459,E2 205.7711} C_DIS
LIN {X -56.346,Y -120.3748,Z 154,A -117.1215,B 22.897,C -0.9627,E1 22.8497,E2 204.2838} C_DIS
LIN {X -53.0475,Y -121.8634,Z 154,A -115.6014,B 22.8972,C -0.9591,E1 22.8536,E2 202.769} C_DIS
LIN {X -50.4557,Y -122.9614,Z 154,A -114.4118,B 22.8972,C -0.9567,E1 22.8566,E2 201.5826} C_DIS
LIN {X -46.9919,Y -124.3243,Z 154,A -112.968,B 22.8976,C -0.9476,E1 22.8603,E2 200.1588} C_DIS
LIN {X -44.3079,Y -125.308,Z 154,A -111.4285,B 22.8971,C -0.961,E1 22.8645,E2 198.5816} C_DIS
LIN {X -41.2179,Y -126.3581,Z 154,A -110.1643,B 22.8974,C -0.9531,E1 22.8678,E2 197.3352} C_DIS
LIN {X -37.6098,Y -127.4763,Z 154,A -108.5294,B 22.8974,C -0.9522,E1 22.8722,E2 195.6994} C_DIS
LIN {X -35.0212,Y -128.2139,Z 154,A -107.375,B 22.8974,C -0.9511,E1 22.8753,E2 194.5458} C_DIS
LIN {X -31.9205,Y -129.0208,Z 154,A -105.8994,B 22.8974,C -0.9548,E1 22.8793,E2 193.0584} C_DIS
LIN {X -28.2593,Y -129.8696,Z 154,A -104.3489,B 22.8974,C -0.9507,E1 22.8835,E2 191.5163} C_DIS
LIN {X -25.099,Y -130.5172,Z 154,A -102.9973,B 22.8976,C -0.9483,E1 22.8872,E2 190.1692} C_DIS
LIN {X -21.1043,Y -131.2246,Z 154,A -101.237,B 22.8976,C -0.9483,E1 22.892,E2 188.4073} C_DIS
LIN {X -18.0354,Y -131.6815,Z 154,A -99.744,B 22.8973,C -0.9553,E1 22.8962,E2 186.8946} C_DIS
LIN {X -14.432,Y -132.1229,Z 154,A -98.2988,B 22.8975,C -0.9494,E1 22.9002,E2 185.4638} C_DIS
LIN {X -10.9804,Y -132.4545,Z 154,A -96.7854,B 22.8975,C -0.9502,E1 22.9044,E2 183.9475} C_DIS
LIN {X -7.0127,Y -132.724,Z 154,A -95.1008,B 22.8975,C -0.9487,E1 22.9091,E2 182.266} C_DIS
LIN {X -3.7186,Y -132.8567,Z 154,A -93.6729,B 22.8975,C -0.9492,E1 22.9131,E2 180.8366} C_DIS
LIN {X 0,Y -132.9108,Z 154,A -91.9444,B 22.8973,C -0.9556,E1 22.9179,E2 179.0918} C_DIS
LIN {X 0,Y -132.9108,Z 154,A -91.9444,B 22.8973,C -0.9556,E1 22.9179,E2 179.0918} C_DIS
Enddeposition()
LIN {X 0.9266,Y -131.9675,Z 154,A -91.3454,B 21.8454,C -0.7909,E1 21.8616,E2 178.8026} C_DIS
Startdeposition()
$VEL.CP = VEL_PRINT
LIN {X -2.9286,Y -131.9406,Z 154,A -93.8073,B 21.8466,C -0.7548,E1 21.8544,E2 181.3616} C_DIS
LIN {X -6.76,Y -131.7979,Z 154,A -95.3879,B 21.8465,C -0.7585,E1 21.85,E2 182.9327} C_DIS
LIN {X -10.8748,Y -131.5224,Z 154,A -97.1208,B 21.8464,C -0.7611,E1 21.8452,E2 184.6592} C_DIS
LIN {X -14.2827,Y -131.1959,Z 154,A -98.6561,B 21.8464,C -0.7591,E1 21.8409,E2 186.201} C_DIS
LIN {X -19.0922,Y -130.5833,Z 154,A -101.0138,B 21.8468,C -0.7483,E1 21.8343,E2 188.5897} C_DIS
LIN {X -24.4222,Y -129.6919,Z 154,A -103.1186,B 21.8464,C -0.7599,E1 21.8286,E2 190.6659} C_DIS
LIN {X -27.8108,Y -129.0072,Z 154,A -104.6127,B 21.8464,C -0.7609,E1 21.8245,E2 192.1594} C_DIS
LIN {X -31.5885,Y -128.1363,Z 154,A -106.2677,B 21.8464,C -0.763,E1 21.82,E2 193.8112} C_DIS
LIN {X -36.3713,Y -126.8619,Z 154,A -109.0084,B 21.8471,C -0.7384,E1 21.8125,E2 196.623} C_DIS
LIN {X -40.9076,Y -125.4729,Z 154,A -110.6102,B 21.8464,C -0.76,E1 21.8084,E2 198.17} C_DIS
LIN {X -44.4347,Y -124.2656,Z 154,A -112.1395,B 21.8462,C -0.7654,E1 21.8044,E2 199.6884} C_DIS
LIN {X -47.6199,Y -123.0798,Z 154,A -113.5856,B 21.8462,C -0.7681,E1 21.8006,E2 201.1308} C_DIS
LIN {X -52.6011,Y -121.0348,Z 154,A -115.9551,B 21.8462,C -0.7691,E1 21.7945,E2 203.5037} C_DIS
LIN {X -56.4288,Y -119.2991,Z 154,A -117.7853,B 21.846,C -0.771,E1 21.7898,E2 205.3342} C_DIS
LIN {X -59.2128,Y -117.9432,Z 154,A -119.1012,B 21.846,C -0.7739,E1 21.7866,E2 206.6463} C_DIS
LIN {X -63.5663,Y -115.6557,Z 154,A -121.3683,B 21.846,C -0.771,E1 21.7809,E2 208.9286} C_DIS
LIN {X -67.4398,Y -113.44,Z 154,A -123.0336,B 21.8455,C -0.7855,E1 21.777,E2 210.5604} C_DIS
LIN {X -70.5971,Y -111.5025,Z 154,A -124.8752,B 21.8458,C -0.7779,E1 21.7726,E2 212.4293} C_DIS
LIN {X -74.2826,Y -109.0824,Z 154,A -126.8431,B 21.8458,C -0.7787,E1 21.768,E2 214.4027} C_DIS
LIN {X -77.0728,Y -107.1292,Z 154,A -128.3361,B 21.8458,C -0.7805,E1 21.7646,E2 215.8967} C_DIS
LIN {X -80.6441,Y -104.4669,Z 154,A -130.2184,B 21.8455,C -0.7862,E1 21.7604,E2 217.7716} C_DIS
LIN {X -83.9242,Y -101.8507,Z 154,A -132.0588,B 21.8455,C -0.7888,E1 21.7564,E2 219.613} C_DIS
LIN {X -87.195,Y -99.0648,Z 154,A -133.9545,B 21.8454,C -0.7911,E1 21.7524,E2 221.5111} C_DIS
LIN {X -90.4109,Y -96.1386,Z 154,A -135.8297,B 21.8452,C -0.7954,E1 21.7486,E2 223.3834} C_DIS
LIN {X -93.1879,Y -93.4494,Z 154,A -137.5587,B 21.8452,C -0.7968,E1 21.7451,E2 225.1171} C_DIS
LIN {X -96.2498,Y -90.2931,Z 154,A -139.4267,B 21.845,C -0.8027,E1 21.7415,E2 226.9786} C_DIS
LIN {X -99.1333,Y -87.1176,Z 154,A -141.3563,B 21.845,C -0.8041,E1 21.7379,E2 228.9146} C_DIS
LIN {X -101.6782,Y -84.1325,Z 154,A -142.997,B 21.8447,C -0.8107,E1 21.735,E2 230.5462} C_DIS
LIN {X -104.296,Y -80.8646,Z 154,A -144.8333,B 21.8445,C -0.8142,E1 21.7318,E2 232.3829} C_DIS
LIN {X -106.8341,Y -77.4803,Z 154,A -146.7059,B 21.8445,C -0.8172,E1 21.7287,E2 234.2579} C_DIS
LIN {X -109.3494,Y -73.8882,Z 154,A -148.5754,B 21.8442,C -0.8235,E1 21.7258,E2 236.1213} C_DIS
LIN {X -112.0939,Y -69.6542,Z 154,A -150.83,B 21.8442,C -0.8265,E1 21.7224,E2 238.3811} C_DIS
LIN {X -114.3646,Y -65.8602,Z 154,A -153.1942,B 21.8446,C -0.8131,E1 21.719,E2 240.7956} C_DIS
LIN {X -116.4777,Y -62.0466,Z 154,A -154.7153,B 21.8439,C -0.8337,E1 21.717,E2 242.2705} C_DIS
LIN {X -118.264,Y -58.5651,Z 154,A -156.3199,B 21.8435,C -0.8423,E1 21.715,E2 243.8618} C_DIS
LIN {X -120.1986,Y -54.4881,Z 154,A -158.535,B 21.8437,C -0.8372,E1 21.7124,E2 246.1047} C_DIS
LIN {X -122.2897,Y -49.6141,Z 154,A -160.4399,B 21.8429,C -0.8604,E1 21.7104,E2 247.9594} C_DIS
LIN {X -125.1365,Y -41.9186,Z 154,A -164.131,B 21.8427,C -0.8654,E1 21.7069,E2 251.6611} C_DIS
LIN {X -126.1458,Y -38.7754,Z 154,A -165.6262,B 21.8427,C -0.8672,E1 21.7056,E2 253.1615} C_DIS
LIN {X -127.0773,Y -35.604,Z 154,A -167.044,B 21.8424,C -0.8722,E1 21.7045,E2 254.5753} C_DIS
LIN {X -127.9367,Y -32.3802,Z 154,A -168.4529,B 21.8422,C -0.8783,E1 21.7035,E2 255.9773} C_DIS
LIN {X -128.7424,Y -29.0145,Z 154,A -170.1358,B 21.8422,C -0.8754,E1 21.7024,E2 257.6793} C_DIS
LIN {X -129.6273,Y -24.7599,Z 154,A -171.9008,B 21.8419,C -0.8863,E1 21.7015,E2 259.4271} C_DIS
LIN {X -130.2763,Y -21.0904,Z 154,A -173.5066,B 21.8417,C -0.8918,E1 21.7007,E2 261.0291} C_DIS
LIN {X -131.1807,Y -14.4238,Z 154,A -176.5512,B 21.8415,C -0.8959,E1 21.6996,E2 264.0837} C_DIS
LIN {X -131.7346,Y -7.8992,Z 154,A -179.2721,B 21.841,C -0.9099,E1 21.699,E2 266.7858} C_DIS
LIN {X -131.9665,Y -1.253,Z 154,A 177.7556,B 21.8407,C -0.9156,E1 21.6988,E2 269.7636} C_DIS
LIN {X -131.9042,Y 4.2388,Z 154,A 175.1964,B 21.8407,C -0.916,E1 21.6989,E2 272.3395} C_DIS
LIN {X -131.7164,Y 8.194,Z 154,A 173.5594,B 21.8404,C -0.9249,E1 21.6991,E2 273.9638} C_DIS
LIN {X -131.4184,Y 12.0759,Z 154,A 171.845,B 21.8402,C -0.9293,E1 21.6995,E2 275.6783} C_DIS
LIN {X -130.7891,Y 17.6285,Z 154,A 169.3127,B 21.84,C -0.9328,E1 21.7004,E2 278.219} C_DIS
LIN {X -130.3053,Y 20.9135,Z 154,A 167.4806,B 21.8405,C -0.9214,E1 21.7012,E2 280.0944} C_DIS
LIN {X -129.5824,Y 24.9949,Z 154,A 166.1309,B 21.8395,C -0.9455,E1 21.7019,E2 281.3883} C_DIS
LIN {X -128.7167,Y 29.127,Z 154,A 164.3076,B 21.8393,C -0.9517,E1 21.703,E2 283.2074} C_DIS
LIN {X -127.9332,Y 32.3943,Z 154,A 162.8691,B 21.839,C -0.9571,E1 21.7039,E2 284.641} C_DIS
LIN {X -127.067,Y 35.6406,Z 154,A 161.4647,B 21.8388,C -0.9639,E1 21.705,E2 286.0365} C_DIS
LIN {X -126.3351,Y 38.1567,Z 154,A 160.3638,B 21.8385,C -0.9689,E1 21.7058,E2 287.1312} C_DIS
LIN {X -125.2934,Y 41.4473,Z 154,A 158.7047,B 21.8386,C -0.967,E1 21.7073,E2 288.8065} C_DIS
LIN {X -124.1621,Y 44.7215,Z 154,A 157.2904,B 21.8383,C -0.9753,E1 21.7085,E2 290.2078} C_DIS
LIN {X -123.0804,Y 47.6182,Z 154,A 155.9594,B 21.8381,C -0.9798,E1 21.7099,E2 291.5352} C_DIS
LIN {X -122.0819,Y 50.1278,Z 154,A 154.5532,B 21.8383,C -0.9738,E1 21.7114,E2 292.9668} C_DIS
LIN {X -120.5465,Y 53.7103,Z 154,A 153.0029,B 21.8379,C -0.9847,E1 21.7131,E2 294.4975} C_DIS
LIN {X -118.6926,Y 57.6964,Z 154,A 150.9171,B 21.8379,C -0.9831,E1 21.7156,E2 296.601} C_DIS
LIN {X -116.9476,Y 61.1516,Z 154,A 149.3477,B 21.8375,C -0.9926,E1 21.7176,E2 298.1544} C_DIS
LIN {X -114.8539,Y 65.0036,Z 154,A 147.3349,B 21.8375,C -0.9935,E1 21.7203,E2 300.1769} C_DIS
LIN {X -112.7382,Y 68.6073,Z 154,A 145.5651,B 21.8372,C -1.0005,E1 21.7228,E2 301.9385} C_DIS
LIN {X -110.4343,Y 72.2575,Z 154,A 143.6162,B 21.8371,C -1.0026,E1 21.7258,E2 303.8931} C_DIS
LIN {X -107.9873,Y 75.8653,Z 154,A 141.704,B 21.8369,C -1.007,E1 21.7288,E2 305.8045} C_DIS
LIN {X -105.2352,Y 79.6386,Z 154,A 139.7294,B 21.8366,C -1.0146,E1 21.7321,E2 307.7696} C_DIS
LIN {X -102.5448,Y 83.0745,Z 154,A 137.7689,B 21.8365,C -1.0168,E1 21.7355,E2 309.7349} C_DIS
LIN {X -99.7311,Y 86.4327,Z 154,A 135.8748,B 21.8362,C -1.022,E1 21.7389,E2 311.625} C_DIS
LIN {X -96.9639,Y 89.5256,Z 154,A 134.0502,B 21.8361,C -1.0255,E1 21.7423,E2 313.4494} C_DIS
LIN {X -93.8953,Y 92.7392,Z 154,A 132.1022,B 21.8359,C -1.0294,E1 21.7461,E2 315.3968} C_DIS
LIN {X -90.7631,Y 95.8064,Z 154,A 130.1975,B 21.8357,C -1.0338,E1 21.75,E2 317.2988} C_DIS
LIN {X -87.5585,Y 98.7435,Z 154,A 128.2948,B 21.8356,C -1.0374,E1 21.7539,E2 319.2005} C_DIS
LIN {X -84.1781,Y 101.6404,Z 154,A 126.3966,B 21.8353,C -1.0431,E1 21.7579,E2 321.0919} C_DIS
LIN {X -80.8647,Y 104.2959,Z 154,A 124.5244,B 21.8352,C -1.0458,E1 21.762,E2 322.9648} C_DIS
LIN {X -77.2851,Y 106.9756,Z 154,A 122.594,B 21.835,C -1.0502,E1 21.7664,E2 324.8914} C_DIS
LIN {X -73.8185,Y 109.3966,Z 154,A 120.8838,B 21.8346,C -1.059,E1 21.7703,E2 326.5843} C_DIS
LIN {X -70.7785,Y 111.388,Z 154,A 119.0961,B 21.8348,C -1.0532,E1 21.7745,E2 328.3946} C_DIS
LIN {X -66.9662,Y 113.7202,Z 154,A 117.166,B 21.8347,C -1.0571,E1 21.7791,E2 330.321} C_DIS
LIN {X -63.2011,Y 115.8549,Z 154,A 115.4482,B 21.8342,C -1.0671,E1 21.7833,E2 332.0176} C_DIS
LIN {X -60.3159,Y 117.3817,Z 154,A 114.0987,B 21.8339,C -1.0723,E1 21.7866,E2 333.3574} C_DIS
LIN {X -56.129,Y 119.4421,Z 154,A 111.369,B 21.8352,C -1.0456,E1 21.7937,E2 336.1673} C_DIS
LIN {X -52.0729,Y 121.2631,Z 154,A 109.3108,B 21.8352,C -1.043,E1 21.799,E2 338.2381} C_DIS
LIN {X -47.2059,Y 123.2407,Z 154,A 107.6301,B 21.834,C -1.0714,E1 21.8032,E2 339.8464} C_DIS
LIN {X -43.4112,Y 124.6265,Z 154,A 106.0646,B 21.8335,C -1.0816,E1 21.8072,E2 341.3879} C_DIS
LIN {X -40.3631,Y 125.6468,Z 154,A 104.5854,B 21.8336,C -1.0796,E1 21.8111,E2 342.8756} C_DIS
LIN {X -37.8352,Y 126.4331,Z 154,A 103.1293,B 21.8342,C -1.0677,E1 21.8151,E2 344.3667} C_DIS
LIN {X -33.9849,Y 127.5198,Z 154,A 101.5629,B 21.8337,C -1.0768,E1 21.8193,E2 345.9114} C_DIS
LIN {X -26.9618,Y 129.189,Z 154,A 98.4226,B 21.8337,C -1.0792,E1 21.8278,E2 349.0499} C_DIS
LIN {X -20.9586,Y 130.2983,Z 154,A 95.7287,B 21.8337,C -1.0792,E1 21.8353,E2 351.747} C_DIS
LIN {X -17.1635,Y 130.8501,Z 154,A 94.2281,B 21.8332,C -1.0874,E1 21.8393,E2 353.2269} C_DIS
LIN {X -13.5193,Y 131.278,Z 154,A 92.6957,B 21.8331,C -1.0908,E1 21.8436,E2 354.7511} C_DIS
LIN {X -10.4774,Y 131.5554,Z 154,A 91.1764,B 21.8334,C -1.083,E1 21.8479,E2 356.2924} C_DIS
LIN {X -6.5917,Y 131.8063,Z 154,A 89.58,B 21.8332,C -1.0877,E1 21.8523,E2 357.8767} C_DIS
LIN {X -2.667,Y 131.945,Z 154,A 87.9908,B 21.833,C -1.0932,E1 21.8567,E2 359.4512} C_DIS
LIN {X 0.6469,Y 131.9696,Z 154,A 86.4319,B 21.8332,C -1.0882,E1 21.8611,E2 361.0237} C_DIS
LIN {X 3.5014,Y 131.9247,Z 154,A 85.0659,B 21.8335,C -1.0827,E1 21.8649,E2 362.404} C_DIS
LIN {X 7.9518,Y 131.7313,Z 154,A 83.2517,B 21.8332,C -1.088,E1 21.8699,E2 364.2033} C_DIS
LIN {X 11.5413,Y 131.4661,Z 154,A 81.7177,B 21.8332,C -1.0891,E1 21.8742,E2 365.7333} C_DIS
LIN {X 15.059,Y 131.1102,Z 154,A 80.0187,B 21.8335,C -1.0816,E1 21.879,E2 367.4513} C_DIS
LIN {X 19.7567,Y 130.4844,Z 154,A 78.0549,B 21.8333,C -1.0852,E1 21.8844,E2 369.4035} C_DIS
LIN {X 23.3111,Y 129.8957,Z 154,A 76.5914,B 21.8332,C -1.0891,E1 21.8884,E2 370.8546} C_DIS
LIN {X 26.6664,Y 129.2491,Z 154,A 75.0425,B 21.8333,C -1.0855,E1 21.8926,E2 372.4111} C_DIS
LIN {X 29.5116,Y 128.6288,Z 154,A 73.6131,B 21.8337,C -1.0774,E1 21.8966,E2 373.8598} C_DIS
LIN {X 33.8172,Y 127.5645,Z 154,A 71.29,B 21.8346,C -1.0584,E1 21.903,E2 376.2297} C_DIS
LIN {X 38.3389,Y 126.2794,Z 154,A 69.835,B 21.8334,C -1.0831,E1 21.9067,E2 377.6155} C_DIS
LIN {X 41.5085,Y 125.2731,Z 154,A 68.3805,B 21.8335,C -1.0814,E1 21.9105,E2 379.0714} C_DIS
LIN {X 44.6283,Y 124.1957,Z 154,A 66.9778,B 21.8335,C -1.0814,E1 21.9142,E2 380.4706} C_DIS
LIN {X 47.3998,Y 123.1653,Z 154,A 65.4802,B 21.834,C -1.0705,E1 21.9182,E2 381.9938} C_DIS
LIN {X 52.008,Y 121.2912,Z 154,A 63.5412,B 21.8337,C -1.0782,E1 21.9231,E2 383.9069} C_DIS
LIN {X 55.1425,Y 119.8983,Z 154,A 61.8453,B 21.8342,C -1.0671,E1 21.9275,E2 385.6276} C_DIS
LIN {X 58.2891,Y 118.4002,Z 154,A 60.1899,B 21.8346,C -1.0587,E1 21.9317,E2 387.3004} C_DIS
LIN {X 61.3816,Y 116.8269,Z 154,A 59.0583,B 21.8339,C -1.0738,E1 21.9344,E2 388.3879} C_DIS
LIN {X 65.0236,Y 114.8426,Z 154,A 57.0298,B 21.8345,C -1.0608,E1 21.9394,E2 390.4443} C_DIS
LIN {X 69.3231,Y 112.2995,Z 154,A 54.9485,B 21.8345,C -1.0615,E1 21.9444,E2 392.5162} C_DIS
LIN {X 73.0967,Y 109.8802,Z 154,A 53.0808,B 21.8345,C -1.062,E1 21.9487,E2 394.3754} C_DIS
LIN {X 76.5312,Y 107.5164,Z 154,A 51.2241,B 21.8347,C -1.0568,E1 21.953,E2 396.2386} C_DIS
LIN {X 80.0999,Y 104.8845,Z 154,A 49.3325,B 21.8347,C -1.0549,E1 21.9572,E2 398.1273} C_DIS
LIN {X 83.6498,Y 102.0758,Z 154,A 47.2812,B 21.8351,C -1.0473,E1 21.9617,E2 400.1902} C_DIS
LIN {X 87.1305,Y 99.1214,Z 154,A 44.5253,B 21.8369,C -1.0077,E1 21.9677,E2 403.0392} C_DIS
LIN {X 92.0437,Y 94.5769,Z 154,A 42.5181,B 21.8353,C -1.0431,E1 21.9715,E2 404.9421} C_DIS
LIN {X 95.0941,Y 91.5096,Z 154,A 40.6214,B 21.8355,C -1.0381,E1 21.9752,E2 406.8427} C_DIS
LIN {X 97.8431,Y 88.5634,Z 154,A 38.8717,B 21.8357,C -1.0342,E1 21.9785,E2 408.5939} C_DIS
LIN {X 100.2343,Y 85.848,Z 154,A 36.7624,B 21.837,C -1.0055,E1 21.9825,E2 410.7688} C_DIS
LIN {X 103.5125,Y 81.8661,Z 154,A 35.0707,B 21.8361,C -1.0256,E1 21.9853,E2 412.3975} C_DIS
LIN {X 106.2278,Y 78.3098,Z 154,A 33.1752,B 21.8361,C -1.0231,E1 21.9885,E2 414.2894} C_DIS
LIN {X 109.0279,Y 74.3626,Z 154,A 31.0916,B 21.8364,C -1.0186,E1 21.9918,E2 416.373} C_DIS
LIN {X 111.3556,Y 70.8295,Z 154,A 29.2327,B 21.8367,C -1.0128,E1 21.9946,E2 418.2366} C_DIS
LIN {X 113.6618,Y 67.0657,Z 154,A 27.3384,B 21.8368,C -1.0087,E1 21.9974,E2 420.1305} C_DIS
LIN {X 115.9275,Y 63.0681,Z 154,A 25.3705,B 21.837,C -1.0046,E1 22,E2 422.0975} C_DIS
LIN {X 117.5188,Y 60.0464,Z 154,A 24.1178,B 21.8367,C -1.0115,E1 22.0016,E2 423.3242} C_DIS
LIN {X 118.5827,Y 57.9191,Z 154,A 22.4807,B 21.8381,C -0.9799,E1 22.0037,E2 425.0354} C_DIS
LIN {X 120.3598,Y 54.1277,Z 154,A 21.1566,B 21.8373,C -0.9981,E1 22.0052,E2 426.3025} C_DIS
LIN {X 121.6787,Y 51.094,Z 154,A 19.7951,B 21.8373,C -0.9976,E1 22.0067,E2 427.6568} C_DIS
LIN {X 122.9615,Y 47.9242,Z 154,A 18.2837,B 21.8376,C -0.992,E1 22.0082,E2 429.1735} C_DIS
LIN {X 124.1501,Y 44.7549,Z 154,A 16.7911,B 21.8378,C -0.9865,E1 22.0097,E2 430.6709} C_DIS
LIN {X 125.2356,Y 41.6211,Z 154,A 15.3661,B 21.8379,C -0.983,E1 22.011,E2 432.0961} C_DIS
LIN {X 126.3313,Y 38.1692,Z 154,A 13.8902,B 21.8379,C -0.9828,E1 22.0122,E2 433.5626} C_DIS
LIN {X 127.346,Y 34.6367,Z 154,A 12.235,B 21.8383,C -0.9751,E1 22.0134,E2 435.2274} C_DIS
LIN {X 129.2932,Y 26.4497,Z 154,A 8.353,B 21.8392,C -0.9529,E1 22.0159,E2 439.1424} C_DIS
LIN {X 130.1808,Y 21.6627,Z 154,A 6.5236,B 21.8389,C -0.9599,E1 22.0168,E2 440.9408} C_DIS
LIN {X 130.72,Y 18.1353,Z 154,A 4.8474,B 21.8394,C -0.949,E1 22.0174,E2 442.6347} C_DIS
LIN {X 131.2325,Y 13.9427,Z 154,A 3.0355,B 21.8396,C -0.9442,E1 22.018,E2 444.4468} C_DIS
LIN {X 131.6144,Y 9.6959,Z 154,A 1.2868,B 21.8396,C -0.9433,E1 22.0184,E2 446.1861} C_DIS
LIN {X 131.8267,Y 6.1866,Z 154,A -0.1647,B 21.8396,C -0.942,E1 22.0186,E2 447.631} C_DIS
LIN {X 131.9458,Y 2.6185,Z 154,A -1.7912,B 21.84,C -0.9333,E1 22.0188,E2 449.2694} C_DIS
LIN {X 131.9681,Y -1.0113,Z 154,A -3.4413,B 21.8404,C -0.9247,E1 22.0188,E2 450.9311} C_DIS
LIN {X 131.8644,Y -5.3063,Z 154,A -5.182,B 21.8404,C -0.9247,E1 22.0186,E2 452.6597} C_DIS
LIN {X 131.6299,Y -9.4834,Z 154,A -7.0252,B 21.8407,C -0.9176,E1 22.0183,E2 454.5092} C_DIS
LIN {X 131.106,Y -15.0945,Z 154,A -9.4501,B 21.8409,C -0.9108,E1 22.0176,E2 456.9357} C_DIS
LIN {X 130.6483,Y -18.6374,Z 154,A -10.8993,B 21.8409,C -0.9108,E1 22.017,E2 458.3751} C_DIS
LIN {X 130.1787,Y -21.6755,Z 154,A -12.3178,B 21.8413,C -0.9024,E1 22.0164,E2 459.806} C_DIS
LIN {X 129.3862,Y -25.9925,Z 154,A -14.1571,B 21.8413,C -0.8995,E1 22.0155,E2 461.6406} C_DIS
LIN {X 128.1329,Y -31.6026,Z 154,A -16.743,B 21.8418,C -0.8873,E1 22.0138,E2 464.2417} C_DIS
LIN {X 127.2701,Y -34.9145,Z 154,A -18.9092,B 21.8432,C -0.8501,E1 22.0122,E2 466.4927} C_DIS
LIN {X 125.5907,Y -40.5389,Z 154,A -20.7618,B 21.8423,C -0.8754,E1 22.0107,E2 468.2657} C_DIS
LIN {X 124.2743,Y -44.4104,Z 154,A -22.3447,B 21.8422,C -0.8791,E1 22.0092,E2 469.8282} C_DIS
LIN {X 123.059,Y -47.6733,Z 154,A -24.2811,B 21.8431,C -0.8542,E1 22.0072,E2 471.8189} C_DIS
LIN {X 121.655,Y -51.1506,Z 154,A -25.5506,B 21.8426,C -0.8664,E1 22.0059,E2 473.0476} C_DIS
LIN {X 119.97,Y -54.9874,Z 154,A -27.3482,B 21.8428,C -0.8619,E1 22.0039,E2 474.8457} C_DIS
LIN {X 118.7067,Y -57.6677,Z 154,A -28.7301,B 21.8431,C -0.8535,E1 22.0022,E2 476.2415} C_DIS
LIN {X 116.1288,Y -62.6969,Z 154,A -31.121,B 21.8433,C -0.8493,E1 21.9991,E2 478.6289} C_DIS
LIN {X 113.9841,Y -66.5169,Z 154,A -33.0056,B 21.8435,C -0.8447,E1 21.9965,E2 480.5146} C_DIS
LIN {X 111.7603,Y -70.1887,Z 154,A -34.8905,B 21.8437,C -0.8384,E1 21.9937,E2 482.4051} C_DIS
LIN {X 109.2581,Y -74.0229,Z 154,A -36.8123,B 21.8437,C -0.836,E1 21.9907,E2 484.3222} C_DIS
LIN {X 106.4557,Y -77.9996,Z 154,A -39.9025,B 21.8456,C -0.784,E1 21.9855,E2 487.5339} C_DIS
LIN {X 102.0316,Y -83.7039,Z 154,A -41.7863,B 21.8438,C -0.8349,E1 21.9824,E2 489.2717} C_DIS
LIN {X 96.938,Y -89.5532,Z 154,A -45.8175,B 21.8452,C -0.7948,E1 21.9748,E2 493.3889} C_DIS
LIN {X 93.8947,Y -92.7397,Z 154,A -47.3233,B 21.8447,C -0.8094,E1 21.9719,E2 494.8484} C_DIS
LIN {X 90.8183,Y -95.7543,Z 154,A -49.0841,B 21.8447,C -0.8101,E1 21.9684,E2 496.5987} C_DIS
LIN {X 87.6187,Y -98.6903,Z 154,A -51.5169,B 21.8457,C -0.78,E1 21.9632,E2 499.1006} C_DIS
LIN {X 84.0569,Y -101.7408,Z 154,A -53.0518,B 21.8451,C -0.799,E1 21.96,E2 500.5778} C_DIS
LIN {X 79.376,Y -105.4334,Z 154,A -56.0331,B 21.8459,C -0.7751,E1 21.9533,E2 503.6104} C_DIS
LIN {X 75.9286,Y -107.9426,Z 154,A -57.4474,B 21.8453,C -0.7918,E1 21.9502,E2 504.9743} C_DIS
LIN {X 72.2867,Y -110.415,Z 154,A -59.3753,B 21.8455,C -0.7873,E1 21.9457,E2 506.9067} C_DIS
LIN {X 68.6072,Y -112.7383,Z 154,A -61.2614,B 21.8456,C -0.784,E1 21.9413,E2 508.795} C_DIS
LIN {X 64.8381,Y -114.9469,Z 154,A -63.138,B 21.8456,C -0.7815,E1 21.9367,E2 510.6714} C_DIS
LIN {X 60.6981,Y -117.1855,Z 154,A -65.4146,B 21.8462,C -0.7672,E1 21.931,E2 512.9788} C_DIS
LIN {X 57.6213,Y -118.7294,Z 154,A -66.6649,B 21.8459,C -0.7762,E1 21.928,E2 514.2014} C_DIS
LIN {X 54.1676,Y -120.342,Z 154,A -68.24,B 21.8459,C -0.7774,E1 21.924,E2 515.7686} C_DIS
LIN {X 51.002,Y -121.7171,Z 154,A -69.709,B 21.8459,C -0.7766,E1 21.9202,E2 517.2356} C_DIS
LIN {X 48.4701,Y -122.7493,Z 154,A -70.9867,B 21.846,C -0.7707,E1 21.9169,E2 518.5257} C_DIS
LIN {X 45.0575,Y -124.041,Z 154,A -72.504,B 21.846,C -0.7718,E1 21.9129,E2 520.0365} C_DIS
LIN {X 41.9072,Y -125.1403,Z 154,A -73.9739,B 21.8461,C -0.769,E1 21.909,E2 521.5104} C_DIS
LIN {X 35.2433,Y -127.1781,Z 154,A -76.9539,B 21.8461,C -0.7677,E1 21.9011,E2 524.4878} C_DIS
LIN {X 31.2585,Y -128.2159,Z 154,A -78.7427,B 21.8462,C -0.7659,E1 21.8962,E2 526.2783} C_DIS
LIN {X 27.1161,Y -129.1572,Z 154,A -80.8291,B 21.8466,C -0.7532,E1 21.8904,E2 528.3958} C_DIS
LIN {X 21.9673,Y -130.13,Z 154,A -82.6652,B 21.846,C -0.7715,E1 21.8855,E2 530.1802} C_DIS
LIN {X 18.2421,Y -130.7047,Z 154,A -84.5603,B 21.8465,C -0.7586,E1 21.8802,E2 532.108} C_DIS
LIN {X 14.2778,Y -131.1964,Z 154,A -86.2118,B 21.8464,C -0.7613,E1 21.8756,E2 533.7507} C_DIS
LIN {X 11.1357,Y -131.5003,Z 154,A -87.634,B 21.8464,C -0.7583,E1 21.8717,E2 535.1801} C_DIS
LIN {X 6.7337,Y -131.7992,Z 154,A -89.4886,B 21.8464,C -0.7603,E1 21.8665,E2 537.0284} C_DIS
LIN {X 2.9571,Y -131.9399,Z 154,A -91.2475,B 21.8466,C -0.7544,E1 21.8616,E2 538.8026} C_DIS
LIN {X 2.9571,Y -131.9399,Z 154,A -91.2475,B 21.8466,C -0.7544,E1 21.8616,E2 538.8026} C_DIS
Enddeposition()
LIN {X 0.9184,Y -131.027,Z 154,A -91.2895,B 20.8216,C -0.6367,E1 20.8328,E2 539.0588} C_DIS
Startdeposition()
$VEL.CP = VEL_PRINT
LIN {X 3.962,Y -130.9739,Z 154,A -89.5975,B 20.8211,C -0.6527,E1 20.8376,E2 537.3225} C_DIS
LIN {X 8.159,Y -130.7791,Z 154,A -87.8634,B 20.8213,C -0.6489,E1 20.8424,E2 535.5998} C_DIS
LIN {X 12.8415,Y -130.4029,Z 154,A -85.8797,B 20.8213,C -0.6468,E1 20.8479,E2 533.6234} C_DIS
LIN {X 15.8294,Y -130.074,Z 154,A -84.4053,B 20.8211,C -0.6545,E1 20.852,E2 532.1286} C_DIS
LIN {X 22.1467,Y -129.1494,Z 154,A -81.6426,B 20.8211,C -0.6551,E1 20.8597,E2 529.3675} C_DIS
LIN {X 30.3275,Y -127.4757,Z 154,A -78.2645,B 20.8213,C -0.6461,E1 20.8688,E2 526.0198} C_DIS
LIN {X 39.8803,Y -124.8167,Z 154,A -74.0933,B 20.8214,C -0.6433,E1 20.88,E2 521.865} C_DIS
LIN {X 44.1431,Y -123.3739,Z 154,A -71.7726,B 20.8209,C -0.6613,E1 20.8862,E2 519.4996} C_DIS
LIN {X 47.4414,Y -122.1431,Z 154,A -69.9207,B 20.8204,C -0.6772,E1 20.8912,E2 517.6078} C_DIS
LIN {X 50.66,Y -120.8438,Z 154,A -68.7471,B 20.8208,C -0.664,E1 20.8941,E2 516.4747} C_DIS
LIN {X 53.8219,Y -119.4694,Z 154,A -67.1726,B 20.8206,C -0.6692,E1 20.8981,E2 514.8904} C_DIS
LIN {X 61.3112,Y -115.8047,Z 154,A -63.6019,B 20.8206,C -0.6716,E1 20.907,E2 511.3248} C_DIS
LIN {X 64.9362,Y -113.813,Z 154,A -61.7318,B 20.8204,C -0.6774,E1 20.9116,E2 509.4451} C_DIS
LIN {X 68.8422,Y -111.4944,Z 154,A -59.7189,B 20.8202,C -0.6822,E1 20.9164,E2 507.4264} C_DIS
LIN {X 72.5794,Y -109.0981,Z 154,A -57.8272,B 20.8202,C -0.6837,E1 20.9208,E2 505.5383} C_DIS
LIN {X 76.1791,Y -106.6155,Z 154,A -55.9056,B 20.8201,C -0.6879,E1 20.9252,E2 503.613} C_DIS
LIN {X 80.1924,Y -103.6306,Z 154,A -53.4174,B 20.8195,C -0.7061,E1 20.9309,E2 501.0849} C_DIS
LIN {X 83.2029,Y -101.2301,Z 154,A -52.0512,B 20.8198,C -0.6953,E1 20.9337,E2 499.7554} C_DIS
LIN {X 88.0058,Y -97.0829,Z 154,A -49.5742,B 20.8201,C -0.688,E1 20.9389,E2 497.3107} C_DIS
LIN {X 92.645,Y -92.6671,Z 154,A -46.7751,B 20.8199,C -0.6944,E1 20.9445,E2 494.508} C_DIS
LIN {X 96.9118,Y -88.1944,Z 154,A -44.0742,B 20.8197,C -0.7008,E1 20.9497,E2 491.8034} C_DIS
LIN {X 100.8475,Y -83.6654,Z 154,A -41.5977,B 20.8197,C -0.7008,E1 20.9542,E2 489.3409} C_DIS
LIN {X 104.4461,Y -79.1268,Z 154,A -38.6121,B 20.8188,C -0.728,E1 20.9595,E2 486.2962} C_DIS
LIN {X 106.5449,Y -76.2778,Z 154,A -37.1683,B 20.8188,C -0.7274,E1 20.9618,E2 484.8626} C_DIS
LIN {X 109.1757,Y -72.4631,Z 154,A -35.1847,B 20.8187,C -0.731,E1 20.9649,E2 482.8811} C_DIS
LIN {X 111.3418,Y -69.088,Z 154,A -33.439,B 20.8185,C -0.7355,E1 20.9675,E2 481.1336} C_DIS
LIN {X 113.4945,Y -65.4916,Z 154,A -31.6086,B 20.8183,C -0.7406,E1 20.9701,E2 479.3005} C_DIS
LIN {X 115.61,Y -61.6814,Z 154,A -28.8745,B 20.8168,C -0.7845,E1 20.9739,E2 476.4612} C_DIS
LIN {X 118.4899,Y -55.9474,Z 154,A -27.0402,B 20.8181,C -0.7477,E1 20.9759,E2 474.7419} C_DIS
LIN {X 119.8873,Y -52.8875,Z 154,A -24.5217,B 20.8162,C -0.8007,E1 20.9789,E2 472.092} C_DIS
LIN {X 122.5368,Y -46.4176,Z 154,A -22.5257,B 20.8176,C -0.7606,E1 20.9808,E2 470.2217} C_DIS
LIN {X 123.7265,Y -43.1444,Z 154,A -20.9717,B 20.8174,C -0.7667,E1 20.9822,E2 468.6615} C_DIS
LIN {X 124.8232,Y -39.86,Z 154,A -18.9541,B 20.8164,C -0.7947,E1 20.984,E2 466.5796} C_DIS
LIN {X 126.1309,Y -35.5064,Z 154,A -17.3193,B 20.8168,C -0.7844,E1 20.9852,E2 464.9849} C_DIS
LIN {X 127.1823,Y -31.5411,Z 154,A -15.4699,B 20.8165,C -0.7926,E1 20.9865,E2 463.1258} C_DIS
LIN {X 128.4447,Y -25.917,Z 154,A -13.3381,B 20.8169,C -0.7825,E1 20.9877,E2 461.0373} C_DIS
LIN {X 129.4789,Y -20.1229,Z 154,A -10.6735,B 20.8164,C -0.7948,E1 20.989,E2 458.3573} C_DIS
LIN {X 130.031,Y -16.1894,Z 154,A -8.1769,B 20.8149,C -0.8356,E1 20.9899,E2 455.7648} C_DIS
LIN {X 130.6198,Y -10.4193,Z 154,A -6.5257,B 20.8161,C -0.8025,E1 20.9903,E2 454.2181} C_DIS
LIN {X 130.872,Y -6.5022,Z 154,A -4.7604,B 20.8159,C -0.8103,E1 20.9906,E2 452.4441} C_DIS
LIN {X 131.0051,Y -2.7938,Z 154,A -3.0399,B 20.8155,C -0.8199,E1 20.9906,E2 450.7091} C_DIS
LIN {X 131.032,Y 0.7769,Z 154,A -1.5664,B 20.8155,C -0.8208,E1 20.9906,E2 449.2437} C_DIS
LIN {X 130.9,Y 5.9441,Z 154,A 0.5657,B 20.8155,C -0.8221,E1 20.9906,E2 447.1237} C_DIS
LIN {X 130.698,Y 9.3698,Z 154,A 2.1441,B 20.8151,C -0.8304,E1 20.9902,E2 445.5335} C_DIS
LIN {X 130.2374,Y 14.4259,Z 154,A 4.8227,B 20.814,C -0.8586,E1 20.9894,E2 442.7956} C_DIS
LIN {X 129.7145,Y 18.5431,Z 154,A 6.1629,B 20.8146,C -0.8423,E1 20.989,E2 441.5106} C_DIS
LIN {X 129.0645,Y 22.6329,Z 154,A 8.7043,B 20.8131,C -0.8817,E1 20.9877,E2 438.8773} C_DIS
LIN {X 127.9629,Y 28.2043,Z 154,A 10.009,B 20.8149,C -0.8349,E1 20.987,E2 437.7125} C_DIS
LIN {X 126.651,Y 33.6036,Z 154,A 12.5485,B 20.8144,C -0.8473,E1 20.9854,E2 435.1566} C_DIS
LIN {X 125.6797,Y 37.072,Z 154,A 14.3588,B 20.8138,C -0.8628,E1 20.9839,E2 433.3157} C_DIS
LIN {X 124.8168,Y 39.8799,Z 154,A 15.656,B 20.8137,C -0.8672,E1 20.9828,E2 432.0152} C_DIS
LIN {X 123.7427,Y 43.0977,Z 154,A 17.1325,B 20.8135,C -0.8712,E1 20.9815,E2 430.5375} C_DIS
LIN {X 122.5099,Y 46.4895,Z 154,A 18.7149,B 20.8133,C -0.876,E1 20.98,E2 428.9526} C_DIS
LIN {X 120.7414,Y 50.9052,Z 154,A 20.8767,B 20.8129,C -0.8857,E1 20.9777,E2 426.7782} C_DIS
LIN {X 118.4909,Y 55.9441,Z 154,A 23.376,B 20.8125,C -0.8964,E1 20.9747,E2 424.2656} C_DIS
LIN {X 116.4906,Y 59.9993,Z 154,A 25.2382,B 20.8125,C -0.8966,E1 20.9724,E2 422.4149} C_DIS
LIN {X 114.3587,Y 63.9709,Z 154,A 27.1866,B 20.8123,C -0.9009,E1 20.9698,E2 420.467} C_DIS
LIN {X 112.0556,Y 67.9241,Z 154,A 28.9696,B 20.8125,C -0.8963,E1 20.9673,E2 418.7081} C_DIS
LIN {X 110.1603,Y 70.9574,Z 154,A 30.7315,B 20.8119,C -0.9093,E1 20.9646,E2 416.9207} C_DIS
LIN {X 106.4847,Y 76.362,Z 154,A 33.4595,B 20.8119,C -0.9106,E1 20.9603,E2 414.2055} C_DIS
LIN {X 104.2038,Y 79.4464,Z 154,A 35.2226,B 20.8116,C -0.9186,E1 20.9573,E2 412.4305} C_DIS
LIN {X 101.3353,Y 83.0741,Z 154,A 37.3129,B 20.8112,C -0.9264,E1 20.9536,E2 410.3301} C_DIS
LIN {X 99.1175,Y 85.7083,Z 154,A 38.7205,B 20.8112,C -0.9255,E1 20.9511,E2 408.933} C_DIS
LIN {X 96.159,Y 89.0152,Z 154,A 40.6579,B 20.8111,C -0.9297,E1 20.9474,E2 406.9944} C_DIS
LIN {X 93.2087,Y 92.0998,Z 154,A 42.5381,B 20.8109,C -0.9343,E1 20.9438,E2 405.111} C_DIS
LIN {X 89.5205,Y 95.688,Z 154,A 44.971,B 20.8103,C -0.9472,E1 20.9388,E2 402.6544} C_DIS
LIN {X 87.0373,Y 97.9527,Z 154,A 45.9214,B 20.8112,C -0.9269,E1 20.937,E2 401.7654} C_DIS
LIN {X 84.7754,Y 99.9163,Z 154,A 47.5331,B 20.8105,C -0.9429,E1 20.9335,E2 400.1167} C_DIS
LIN {X 81.666,Y 102.4733,Z 154,A 49.2663,B 20.8105,C -0.945,E1 20.9297,E2 398.3857} C_DIS
LIN {X 78.0249,Y 105.2726,Z 154,A 51.2744,B 20.8103,C -0.9485,E1 20.9252,E2 396.3765} C_DIS
LIN {X 74.4091,Y 107.8587,Z 154,A 53.1867,B 20.8102,C -0.9504,E1 20.9209,E2 394.4669} C_DIS
LIN {X 71.3686,Y 109.8938,Z 154,A 54.7806,B 20.8101,C -0.9527,E1 20.9171,E2 392.873} C_DIS
LIN {X 67.7236,Y 112.1769,Z 154,A 57.1034,B 20.8091,C -0.9751,E1 20.9115,E2 390.4964} C_DIS
LIN {X 63.8744,Y 114.413,Z 154,A 58.5181,B 20.81,C -0.9544,E1 20.9082,E2 389.1448} C_DIS
LIN {X 60.8199,Y 116.0627,Z 154,A 60.0268,B 20.81,C -0.9561,E1 20.9045,E2 387.6367} C_DIS
LIN {X 57.1009,Y 117.9388,Z 154,A 61.9852,B 20.8096,C -0.9644,E1 20.8995,E2 385.6616} C_DIS
LIN {X 53.2349,Y 119.732,Z 154,A 63.6913,B 20.8098,C -0.9597,E1 20.8952,E2 383.9738} C_DIS
LIN {X 49.9505,Y 121.1401,Z 154,A 65.7983,B 20.8086,C -0.9851,E1 20.8896,E2 381.8014} C_DIS
LIN {X 45.8574,Y 122.7467,Z 154,A 67.167,B 20.8096,C -0.9629,E1 20.8862,E2 380.4989} C_DIS
LIN {X 42.8452,Y 123.8302,Z 154,A 68.5829,B 20.8096,C -0.9648,E1 20.8825,E2 379.0809} C_DIS
LIN {X 39.6292,Y 124.8969,Z 154,A 70.0103,B 20.8096,C -0.9637,E1 20.8787,E2 377.66} C_DIS
LIN {X 36.2287,Y 125.9266,Z 154,A 71.8118,B 20.8091,C -0.9756,E1 20.8738,E2 375.829} C_DIS
LIN {X 31.9043,Y 127.0901,Z 154,A 73.5567,B 20.8094,C -0.9677,E1 20.8692,E2 374.1097} C_DIS
LIN {X 27.3671,Y 128.1437,Z 154,A 75.4394,B 20.8097,C -0.9622,E1 20.8641,E2 372.2455} C_DIS
Enddeposition()
END
